// TwinCAT 3 PLC project CNM_AssertionInterfaceTests
// Title: CNM_AssertionInterfaceTests
// Company: ekvip automation GmbH
// Author: boez & ajum
// ProjectVersion: 1.0.0.47
// Description: Foo bar baz
// ProgramVersion: 3.1.4026.16
// libraries:
//   CNM_AbstractObject, * (ekvip automation GmbH)
//   CNM_AssertionInterfaceLib, * (ekvip automation GmbH)
//   CNM_ReturnTypes, * (ekvip automation GmbH)
//   Tc2_CncBase, * (Beckhoff Automation GmbH)
//   Tc2_CncHli, * (Beckhoff Automation GmbH)
//   Tc2_Standard, * (Beckhoff Automation GmbH)
//   Tc2_System, * (Beckhoff Automation GmbH)
//   Tc2_Utilities, * (Beckhoff Automation GmbH)
//   Tc3_Module, * (Beckhoff Automation GmbH)
//   TcUnit, * (www.tcunit.org)
// project tree:
//   AssertionTester/AssertionResult/interfaces/ IAssertorContainer.TcIO
//   AssertionTester/AssertionTests/BinaryAssertions/classes/ BinaryAssertionsTests.TcPOU, gfdfdfdvdfvdfvdfvfdv.TcPOU
//   AssertionTester/AssertionTests/BitNumberAssertions/classes/ XWordAssertionTests.TcPOU
//   AssertionTester/AssertionTests/classes/ AbstractAssertorTest.TcPOU
//   AssertionTester/AssertionTests/DateTimeAssertions/classes/ DTAssertionTests.TcPOU, DateAssertionTests.TcPOU, TODAssertionTests.TcPOU
//   AssertionTester/AssertionTests/FloatAssertions/classes/ RealAssertionTests.TcPOU, LRealAssertionTests.TcPOU
//   AssertionTester/AssertionTests/FloatAssertions/types/structs/ LRealTestParameter.TcDUT
//   AssertionTester/AssertionTests/IntegerAssertions/classes/ DintAssertionTests.TcPOU, IntAssertionTests.TcPOU, LintAssertionTests.TcPOU, SintAssertionTests.TcPOU, UdintAssertionTests.TcPOU, UintAssertionTests.TcPOU, UlintAssertionTests.TcPOU, UsintAssertionTests.TcPOU, UxintAssertionTests.TcPOU, XintAssertionTests.TcPOU
//   AssertionTester/AssertionTests/PointerAssertions/ PointerAssertionsTests.TcPOU
//   AssertionTester/AssertionTests/StringAssertions/InputStructs/common/ AnyTestString.TcDUT, StringType.TcDUT
//   AssertionTester/AssertionTests/StringAssertions/InputStructs/containsStr/ containsDataStr.TcDUT
//   AssertionTester/AssertionTests/StringAssertions/InputStructs/isEmptyStr/ isEmptyDataStr.TcDUT
//   AssertionTester/AssertionTests/StringAssertions/InputStructs/isEqualStr/ isEqualToDataStr.TcDUT
//   AssertionTester/AssertionTests/StringAssertions/InputStructs/isLenghtBetweenStr/ IsLengthBetweenBasicData.TcDUT
//   AssertionTester/AssertionTests/StringAssertions/InputStructs/isLenghtStr/ FunctionType.TcDUT, IsLengthBasicData.TcDUT, StringTestDataIsLength.TcDUT, TypeToTest.TcDUT
//   AssertionTester/AssertionTests/StringAssertions/ StringAssertionTests.TcPOU
//   AssertionTester/AssertionTests/StringAssertions/TestDataSets/ containsNoTestDataSet.TcGVL, containsTestDataSet.TcGVL, endsWithDataSet.TcGVL, isEmptyTestDataSet.TcGVL, isEqualToTestDataSet.TcGVL, IsLengthBetweenDataSet.TcGVL, IsLengthTestDataSet.TcGVL, isNotEmtyTestDataSet.TcGVL, isNotEqualToTestDataSet.TcGVL, startsWithDataSet.TcGVL
//   AssertionTester/AssertionTests/TimeAssertions/ TimeAssertionsTests.TcPOU
//   AssertionTester/classes/ AssertionTester.TcPOU
//   AssertionTester/functions/ ArrayOfMessageStringToString.TcPOU
//   AssertionTester/interfaces/ IAttachAssertorContainer.TcIO
//   Project Information/ F_GetCompany.TcPOU, F_GetTitle.TcPOU, F_GetVersion.TcPOU
//   Version/ Global_Version.TcGVL

// ---- AssertionTester/AssertionTests/FloatAssertions/types/structs/LRealTestParameter.TcDUT
(*

short summary
=================
this is just a helper type, the TwinCAT function LREAL_TO_STRING
throws an exception with the value 2.225073858507201e-308. 
since there is no big integer arithmetic at TwinCAT 
it's not in the scope of the test library to implement a doubleToString.
This data type contains just a LREAL value and it's string representation.

.. <legal notes>

legal notes
=================
| SPDX-FileCopyrightText: © 2022 ekvip automation GmbH <info@ekvip.de>
| SPDX-License-Identifier: Apache-2.0
| For details check: Apache-2.0_

.. _Apache-2.0: https://www.apache.org/licenses/LICENSE-2.0

.. </legal notes>

type members
======================

*)

TYPE LRealTestParameter :
STRUCT
	(* just the value to test *)
	value		:LREAL;
	(* string representation of ``value`` *)
	asString	:Tc2_System.T_MaxString;
END_STRUCT
END_TYPE

// ---- AssertionTester/AssertionTests/StringAssertions/InputStructs/common/AnyTestString.TcDUT
(*

short summary
=============

.. <legal notes>

legal notes
=================
| SPDX-FileCopyrightText: © 2023 ekvip automation GmbH <info@ekvip.de>
| SPDX-License-Identifier: Apache-2.0
| For details check: Apache-2.0_

.. _Apache-2.0: https://www.apache.org/licenses/LICENSE-2.0

.. </legal notes>

*)

{warning 'header is generated please add your documentation'}
TYPE AnyTestString :
STRUCT
	wstringToTest	:WSTRING(300);
	stringToTest	:STRING(600);
END_STRUCT
END_TYPE

// ---- AssertionTester/AssertionTests/StringAssertions/InputStructs/common/StringType.TcDUT
(*

short summary
=============

.. <legal notes>

legal notes
=================
| SPDX-FileCopyrightText: © 2023 ekvip automation GmbH <info@ekvip.de>
| SPDX-License-Identifier: Apache-2.0
| For details check: Apache-2.0_

.. _Apache-2.0: https://www.apache.org/licenses/LICENSE-2.0

.. </legal notes>

enumeration values
==================

*)

{warning 'header is generated please add your documentation'}
{attribute 'qualified_only'}
{attribute 'strict'}
{attribute 'to_string'}
TYPE StringType :
(
	ASCII_STRING := 0,
	UTF16STRING  := 1
)USINT;
END_TYPE

// ---- AssertionTester/AssertionTests/StringAssertions/InputStructs/containsStr/containsDataStr.TcDUT
(*

short summary
=============

.. <legal notes>

legal notes
=================
| SPDX-FileCopyrightText: © 2023 ekvip automation GmbH <info@ekvip.de>
| SPDX-License-Identifier: Apache-2.0
| For details check: Apache-2.0_

.. _Apache-2.0: https://www.apache.org/licenses/LICENSE-2.0

.. </legal notes>

*)

{warning 'header is generated please add your documentation'}
TYPE containsDataStr :
STRUCT
	StringToTest		: STRING;
	WStringToTest 		: WSTRING;
	StringToContain 	: STRING;
	WStringToContain	: WSTRING;
	IgnoreCases			: BOOL;
	Trim 				: BOOL;
	ExpectedResult  	: BOOL;
	typeToTest      	: TypeToTest;		
END_STRUCT
END_TYPE

// ---- AssertionTester/AssertionTests/StringAssertions/InputStructs/isEmptyStr/isEmptyDataStr.TcDUT
(*

short summary
=============

.. <legal notes>

legal notes
=================
| SPDX-FileCopyrightText: © 2023 ekvip automation GmbH <info@ekvip.de>
| SPDX-License-Identifier: Apache-2.0
| For details check: Apache-2.0_

.. _Apache-2.0: https://www.apache.org/licenses/LICENSE-2.0

.. </legal notes>

*)

{warning 'header is generated please add your documentation'}
TYPE isEmptyDataStr :
STRUCT
	StringToTest		: STRING;
	WStringToTest 		: WSTRING;
	ExpectedResult  	: BOOL;
	typeToTest      	: TypeToTest;		
END_STRUCT
END_TYPE

// ---- AssertionTester/AssertionTests/StringAssertions/InputStructs/isEqualStr/isEqualToDataStr.TcDUT
(*

short summary
=============

.. <legal notes>

legal notes
=================
| SPDX-FileCopyrightText: © 2023 ekvip automation GmbH <info@ekvip.de>
| SPDX-License-Identifier: Apache-2.0
| For details check: Apache-2.0_

.. _Apache-2.0: https://www.apache.org/licenses/LICENSE-2.0

.. </legal notes>

*)

{warning 'header is generated please add your documentation'}
TYPE isEqualToDataStr :
STRUCT
	StringToTest		: STRING;
	WStringToTest 		: WSTRING;
	EqualToString		: STRING;
	EqualToWString 		: WSTRING;
	IgnoreCases			: BOOL;
	ExpectedResult  	: BOOL;
	typeToTest      	: TypeToTest;		
END_STRUCT
END_TYPE

// ---- AssertionTester/AssertionTests/StringAssertions/InputStructs/isLenghtBetweenStr/IsLengthBetweenBasicData.TcDUT
(*

short summary
=============

.. <legal notes>

legal notes
=================
| SPDX-FileCopyrightText: © 2023 ekvip automation GmbH <info@ekvip.de>
| SPDX-License-Identifier: Apache-2.0
| For details check: Apache-2.0_

.. _Apache-2.0: https://www.apache.org/licenses/LICENSE-2.0

.. </legal notes>

*)

{warning 'header is generated please add your documentation'}
TYPE IsLengthBetweenBasicData :
STRUCT
	StringToTest	: STRING;
	WStringToTest	: WSTRING;
	ExpectedResult  : BOOL;
	maxLength		: USINT;
	minLength		: USINT; 
	typeToTest      : TypeToTest;  
END_STRUCT
END_TYPE

// ---- AssertionTester/AssertionTests/StringAssertions/InputStructs/isLenghtStr/FunctionType.TcDUT
(*

short summary
=============

.. <legal notes>

legal notes
=================
| SPDX-FileCopyrightText: © 2023 ekvip automation GmbH <info@ekvip.de>
| SPDX-License-Identifier: Apache-2.0
| For details check: Apache-2.0_

.. _Apache-2.0: https://www.apache.org/licenses/LICENSE-2.0

.. </legal notes>

enumeration values
==================

*)

{warning 'header is generated please add your documentation'}
{attribute 'qualified_only'}
{attribute 'strict'}
{attribute 'to_string'}
TYPE FunctionType :
(
	EXACT 	:= 0,
	MAXIMUM := 1,
	MINIMUM	:= 2 
);
END_TYPE

// ---- AssertionTester/AssertionTests/StringAssertions/InputStructs/isLenghtStr/IsLengthBasicData.TcDUT
(*

short summary
=============

.. <legal notes>

legal notes
=================
| SPDX-FileCopyrightText: © 2023 ekvip automation GmbH <info@ekvip.de>
| SPDX-License-Identifier: Apache-2.0
| For details check: Apache-2.0_

.. _Apache-2.0: https://www.apache.org/licenses/LICENSE-2.0

.. </legal notes>

*)

{warning 'header is generated please add your documentation'}
TYPE IsLengthBasicData :
STRUCT
	StringToTest	: STRING;
	WStringToTest	: WSTRING;
	ExpectedResult  : BOOL;
	ExpectedLength	: UDINT; 
	FuncType		: FunctionType;
	typeToTest      : TypeToTest;  	
END_STRUCT
END_TYPE

// ---- AssertionTester/AssertionTests/StringAssertions/InputStructs/isLenghtStr/StringTestDataIsLength.TcDUT
(*

short summary
=============

.. <legal notes>

legal notes
=================
| SPDX-FileCopyrightText: © 2023 ekvip automation GmbH <info@ekvip.de>
| SPDX-License-Identifier: Apache-2.0
| For details check: Apache-2.0_

.. _Apache-2.0: https://www.apache.org/licenses/LICENSE-2.0

.. </legal notes>

*)

{warning 'header is generated please add your documentation'}
TYPE StringTestDataIsLength :
STRUCT
	testString		: AnyTestString ;
	expectedLength	: UDINT;
	stringType		: StringType;
	message			: STRING;
	expectedResult	: BOOL;
    funcType		: FunctionType;     
END_STRUCT
END_TYPE

// ---- AssertionTester/AssertionTests/StringAssertions/InputStructs/isLenghtStr/TypeToTest.TcDUT
(*

short summary
=============

.. <legal notes>

legal notes
=================
| SPDX-FileCopyrightText: © 2023 ekvip automation GmbH <info@ekvip.de>
| SPDX-License-Identifier: Apache-2.0
| For details check: Apache-2.0_

.. _Apache-2.0: https://www.apache.org/licenses/LICENSE-2.0

.. </legal notes>

enumeration values
==================

*)

{warning 'header is generated please add your documentation'}
{attribute 'qualified_only'}
{attribute 'strict'}
TYPE TypeToTest :
(
	TEST_STRING 	:= 0,
	TEST_WSTRING 	:= 1
);
END_TYPE

// ---- AssertionTester/AssertionTests/StringAssertions/TestDataSets/containsNoTestDataSet.TcGVL
(*

short summary
=============

.. <legal notes>

legal notes
=================
| SPDX-FileCopyrightText: © 2023 ekvip automation GmbH <info@ekvip.de>
| SPDX-License-Identifier: Apache-2.0
| For details check: Apache-2.0_

.. _Apache-2.0: https://www.apache.org/licenses/LICENSE-2.0

.. </legal notes>

*)

{warning 'header is generated please add your documentation'}
{attribute 'qualified_only'}
VAR_GLOBAL CONSTANT
	SIZE_OF_CONTAINSNO_DATASET:USINT := 21;
END_VAR

VAR_GLOBAL
	containsNoDataSetCommon : ARRAY[0..SIZE_OF_CONTAINSNO_DATASET] OF containsDataStr := [
		
		// test number 0
		(	StringToTest		:= 'hello',
		  	WStringToTest 		:= "Hello",
			StringToContain 	:= 'h',
			WStringToContain	:= "h",
			IgnoreCases			:= TRUE,
			ExpectedResult  	:= TRUE,
			typeToTest      	:= TypeToTest.TEST_STRING	),
		
		// test number 1	
		(	StringToTest		:= 'hello',
		  	WStringToTest 		:= "Hello",
			StringToContain 	:= 'h',
			WStringToContain	:= "h",
			IgnoreCases			:= TRUE,
			ExpectedResult  	:= TRUE,
			typeToTest      	:= TypeToTest.TEST_WSTRING	),
		
		// test number 2		
		(	StringToTest		:= 'дивный новый мир',
		  	WStringToTest 		:= "дивный новый мир",
			StringToContain 	:= 'нов',
			WStringToContain	:= "нов",
			IgnoreCases			:= TRUE,
			ExpectedResult  	:= TRUE,
			typeToTest      	:= TypeToTest.TEST_WSTRING	),

		// test number 3				
		(	StringToTest		:= 'дивный новый мир',
		  	WStringToTest 		:= "дивный новый мир",
			StringToContain 	:= 'ноa',
			WStringToContain	:= "ноa",
			IgnoreCases			:= TRUE,
			ExpectedResult  	:= FALSE,
			typeToTest      	:= TypeToTest.TEST_WSTRING	),

		// test number 4				
		(	StringToTest		:= 'дивный новый мир',
		  	WStringToTest 		:= "дивный новый мир",
			StringToContain 	:= 'нов',
			WStringToContain	:= "нов",
			IgnoreCases			:= TRUE,
			ExpectedResult  	:= TRUE,
			typeToTest      	:= TypeToTest.TEST_STRING	),
	
		// test number 5			
		(	StringToTest		:= 'дивный новый мир',
		  	WStringToTest 		:= "дивный новый мир",
			StringToContain 	:= 'ноa',
			WStringToContain	:= "ноa",
			IgnoreCases			:= TRUE,
			ExpectedResult  	:= FALSE,
			typeToTest      	:= TypeToTest.TEST_STRING	),
			
		// test number 6			
		(	StringToTest		:= '',
		  	WStringToTest 		:= "",
			StringToContain 	:= ' ',
			WStringToContain	:= " ",
			IgnoreCases			:= TRUE,
			ExpectedResult  	:= FALSE,
			typeToTest      	:= TypeToTest.TEST_STRING	),
			
		// test number 7			
		(	StringToTest		:= '',
		  	WStringToTest 		:= "",
			StringToContain 	:= ' ',
			WStringToContain	:= " ",
			IgnoreCases			:= TRUE,
			ExpectedResult  	:= FALSE,
			typeToTest      	:= TypeToTest.TEST_WSTRING	),
			
		// test number 8			
		(	StringToTest		:= ' ',
		  	WStringToTest 		:= " ",
			StringToContain 	:= ' ',
			WStringToContain	:= " ",
			IgnoreCases			:= TRUE,
			ExpectedResult  	:= TRUE,
			typeToTest      	:= TypeToTest.TEST_STRING	),
			
		// test number 9			
		(	StringToTest		:= ' ',
		  	WStringToTest 		:= " ",
			StringToContain 	:= ' ',
			WStringToContain	:= " ",
			IgnoreCases			:= TRUE,
			ExpectedResult  	:= TRUE,
			typeToTest      	:= TypeToTest.TEST_WSTRING	),
			
		// test number 10			
		(	StringToTest		:= ' ',
		  	WStringToTest 		:= " ",
			StringToContain 	:= ' ',
			WStringToContain	:= " ",
			IgnoreCases			:= TRUE,
			ExpectedResult  	:= TRUE,
			typeToTest      	:= TypeToTest.TEST_STRING	),
			
		// test number 11			
		(	StringToTest		:= 'Brave new World',
		  	WStringToTest 		:= "Brave new World",
			StringToContain 	:= 'brave',
			WStringToContain	:= "brave",
			IgnoreCases			:= FALSE,
			ExpectedResult  	:= FALSE,
			typeToTest      	:= TypeToTest.TEST_WSTRING	),
			
		// test number 12			
		(	StringToTest		:= 'Brave new World',
		  	WStringToTest 		:= "Brave new World",
			StringToContain 	:= 'brave',
			WStringToContain	:= "brave",
			IgnoreCases			:= FALSE,
			ExpectedResult  	:= FALSE,
			typeToTest      	:= TypeToTest.TEST_WSTRING	),
			
		// test number 13			
		(	StringToTest		:= 'Brave new World',
		  	WStringToTest 		:= "Brave new World",
			StringToContain 	:= 'brave',
			WStringToContain	:= "brave",
			IgnoreCases			:= TRUE,
			ExpectedResult  	:= TRUE,
			typeToTest      	:= TypeToTest.TEST_WSTRING	),
			
		// test number 14			
		(	StringToTest		:= 'Brave new World',
		  	WStringToTest 		:= "Brave new World",
			StringToContain 	:= 'brave',
			WStringToContain	:= "brave",
			IgnoreCases			:= TRUE,
			ExpectedResult  	:= TRUE,
			typeToTest      	:= TypeToTest.TEST_WSTRING	),
			
		// test number 15			
		(	StringToTest		:= '²345',
		  	WStringToTest 		:= "²345",
			StringToContain 	:= '2',
			WStringToContain	:= "2",
			IgnoreCases			:= TRUE,
			ExpectedResult  	:= FALSE,
			typeToTest      	:= TypeToTest.TEST_STRING	),
			
		// test number 16			
		(	StringToTest		:= '2345',
		  	WStringToTest 		:= "²345",
			StringToContain 	:= '2',
			WStringToContain	:= "2",
			IgnoreCases			:= TRUE,
			ExpectedResult  	:= FALSE,
			typeToTest      	:= TypeToTest.TEST_WSTRING	),
			
		// test number 17			
		(	StringToTest		:= '²345',
		  	WStringToTest 		:= "²345",
			StringToContain 	:= '2',
			WStringToContain	:= "2",
			IgnoreCases			:= FALSE,
			ExpectedResult  	:= FALSE,
			typeToTest      	:= TypeToTest.TEST_STRING	),
			
		// test number 18			
		(	StringToTest		:= '²345',
		  	WStringToTest 		:= "²345",
			StringToContain 	:= '2',
			WStringToContain	:= "2",
			IgnoreCases			:= FALSE,
			ExpectedResult  	:= FALSE,
			typeToTest      	:= TypeToTest.TEST_WSTRING	),
			
		// test number 19			
		(	StringToTest		:= '',
		  	WStringToTest 		:= "👪",
			StringToContain 	:= '',
			WStringToContain	:= "👪",
			IgnoreCases			:= FALSE,
			ExpectedResult  	:= TRUE,
			typeToTest      	:= TypeToTest.TEST_WSTRING	),
			
		// test number 20			
		(	StringToTest		:= ' hello world ',
		  	WStringToTest 		:= " hello world ",
			StringToContain 	:= '  ',
			WStringToContain	:= "  ",
			IgnoreCases			:= FALSE,
			ExpectedResult  	:= FALSE,
			typeToTest      	:= TypeToTest.TEST_WSTRING	),
			
		// test number 21			
		(	StringToTest		:= ' hello world ',
		  	WStringToTest 		:= " hello world ",
			StringToContain 	:= '  ',
			WStringToContain	:= "  ",
			IgnoreCases			:= FALSE,
			ExpectedResult  	:= FALSE,
			typeToTest      	:= TypeToTest.TEST_STRING	)
			
		
			
		

	];
END_VAR

// ---- AssertionTester/AssertionTests/StringAssertions/TestDataSets/containsTestDataSet.TcGVL
(*

short summary
=============

.. <legal notes>

legal notes
=================
| SPDX-FileCopyrightText: © 2023 ekvip automation GmbH <info@ekvip.de>
| SPDX-License-Identifier: Apache-2.0
| For details check: Apache-2.0_

.. _Apache-2.0: https://www.apache.org/licenses/LICENSE-2.0

.. </legal notes>

*)

{warning 'header is generated please add your documentation'}
{attribute 'qualified_only'}
VAR_GLOBAL CONSTANT
	SIZE_OF_CONTAINS_DATASET:USINT := 23;
END_VAR

VAR_GLOBAL
	containsDataSetCommon : ARRAY[0..SIZE_OF_CONTAINS_DATASET] OF containsDataStr := [
		// test number 0
		(	StringToTest		:= 'hello',
		  	WStringToTest 		:= "Hello",
			StringToContain 	:= 'h',
			WStringToContain	:= "h",
			IgnoreCases			:= TRUE,
			ExpectedResult  	:= FALSE,
			typeToTest      	:= TypeToTest.TEST_STRING	),
		
		// test number 1	
		(	StringToTest		:= 'hello',
		  	WStringToTest 		:= "Hello",
			StringToContain 	:= 'h',
			WStringToContain	:= "h",
			IgnoreCases			:= TRUE,
			ExpectedResult  	:= FALSE,
			typeToTest      	:= TypeToTest.TEST_WSTRING	),
		
		// test number 2		
		(	StringToTest		:= 'дивный новый мир',
		  	WStringToTest 		:= "дивный новый мир",
			StringToContain 	:= 'нов',
			WStringToContain	:= "нов",
			IgnoreCases			:= TRUE,
			ExpectedResult  	:= FALSE,
			typeToTest      	:= TypeToTest.TEST_WSTRING	),

		// test number 3				
		(	StringToTest		:= 'дивный новый мир',
		  	WStringToTest 		:= "дивный новый мир",
			StringToContain 	:= 'ноa',
			WStringToContain	:= "ноa",
			IgnoreCases			:= TRUE,
			ExpectedResult  	:= TRUE,
			typeToTest      	:= TypeToTest.TEST_WSTRING	),

		// test number 4				
		(	StringToTest		:= 'дивный новый мир',
		  	WStringToTest 		:= "дивный новый мир",
			StringToContain 	:= 'нов',
			WStringToContain	:= "нов",
			IgnoreCases			:= TRUE,
			ExpectedResult  	:= FALSE,
			typeToTest      	:= TypeToTest.TEST_STRING	),
	
		// test number 5			
		(	StringToTest		:= 'дивный новый мир',
		  	WStringToTest 		:= "дивный новый мир",
			StringToContain 	:= 'ноa',
			WStringToContain	:= "ноa",
			IgnoreCases			:= TRUE,
			ExpectedResult  	:= TRUE,
			typeToTest      	:= TypeToTest.TEST_STRING	),
			
		// test number 6			
		(	StringToTest		:= '',
		  	WStringToTest 		:= "",
			StringToContain 	:= ' ',
			WStringToContain	:= " ",
			IgnoreCases			:= TRUE,
			ExpectedResult  	:= TRUE,
			typeToTest      	:= TypeToTest.TEST_STRING	),
			
		// test number 7			
		(	StringToTest		:= '',
		  	WStringToTest 		:= "",
			StringToContain 	:= ' ',
			WStringToContain	:= " ",
			IgnoreCases			:= TRUE,
			ExpectedResult  	:= TRUE,
			typeToTest      	:= TypeToTest.TEST_WSTRING	),
			
		// test number 8			
		(	StringToTest		:= ' ',
		  	WStringToTest 		:= " ",
			StringToContain 	:= ' ',
			WStringToContain	:= " ",
			IgnoreCases			:= TRUE,
			ExpectedResult  	:= FALSE,
			typeToTest      	:= TypeToTest.TEST_STRING	),
			
		// test number 9			
		(	StringToTest		:= ' ',
		  	WStringToTest 		:= " ",
			StringToContain 	:= ' ',
			WStringToContain	:= " ",
			IgnoreCases			:= TRUE,
			ExpectedResult  	:= FALSE,
			typeToTest      	:= TypeToTest.TEST_WSTRING	),
			
		// test number 10			
		(	StringToTest		:= ' ',
		  	WStringToTest 		:= " ",
			StringToContain 	:= ' ',
			WStringToContain	:= " ",
			IgnoreCases			:= TRUE,
			ExpectedResult  	:= FALSE,
			typeToTest      	:= TypeToTest.TEST_STRING	),
			
		// test number 11			
		(	StringToTest		:= 'Brave new World',
		  	WStringToTest 		:= "Brave new World",
			StringToContain 	:= 'brave',
			WStringToContain	:= "brave",
			IgnoreCases			:= FALSE,
			ExpectedResult  	:= TRUE,
			typeToTest      	:= TypeToTest.TEST_WSTRING	),
			
		// test number 12			
		(	StringToTest		:= 'Brave new World',
		  	WStringToTest 		:= "Brave new World",
			StringToContain 	:= 'brave',
			WStringToContain	:= "brave",
			IgnoreCases			:= FALSE,
			ExpectedResult  	:= TRUE,
			typeToTest      	:= TypeToTest.TEST_WSTRING	),
			
		// test number 13			
		(	StringToTest		:= 'Brave new World',
		  	WStringToTest 		:= "Brave new World",
			StringToContain 	:= 'brave',
			WStringToContain	:= "brave",
			IgnoreCases			:= TRUE,
			ExpectedResult  	:= FALSE,
			typeToTest      	:= TypeToTest.TEST_WSTRING	),
			
		// test number 14			
		(	StringToTest		:= 'Brave new World',
		  	WStringToTest 		:= "Brave new World",
			StringToContain 	:= 'brave',
			WStringToContain	:= "brave",
			IgnoreCases			:= TRUE,
			ExpectedResult  	:= FALSE,
			typeToTest      	:= TypeToTest.TEST_WSTRING	),
			
		// test number 15			
		(	StringToTest		:= '²345',
		  	WStringToTest 		:= "²345",
			StringToContain 	:= '2',
			WStringToContain	:= "2",
			IgnoreCases			:= TRUE,
			ExpectedResult  	:= TRUE,
			typeToTest      	:= TypeToTest.TEST_STRING	),
			
		// test number 16			
		(	StringToTest		:= '2345',
		  	WStringToTest 		:= "²345",
			StringToContain 	:= '2',
			WStringToContain	:= "2",
			IgnoreCases			:= TRUE,
			ExpectedResult  	:= TRUE,
			typeToTest      	:= TypeToTest.TEST_WSTRING	),
			
		// test number 17			
		(	StringToTest		:= '²345',
		  	WStringToTest 		:= "²345",
			StringToContain 	:= '2',
			WStringToContain	:= "2",
			IgnoreCases			:= FALSE,
			ExpectedResult  	:= TRUE,
			typeToTest      	:= TypeToTest.TEST_STRING	),
			
		// test number 18			
		(	StringToTest		:= '²345',
		  	WStringToTest 		:= "²345",
			StringToContain 	:= '2',
			WStringToContain	:= "2",
			IgnoreCases			:= FALSE,
			ExpectedResult  	:= TRUE,
			typeToTest      	:= TypeToTest.TEST_WSTRING	),
			
		// test number 19			
		(	StringToTest		:= '',
		  	WStringToTest 		:= "👪",
			StringToContain 	:= '',
			WStringToContain	:= "👪",
			IgnoreCases			:= FALSE,
			ExpectedResult  	:= FALSE,
			typeToTest      	:= TypeToTest.TEST_WSTRING	),
			
		// test number 20			
		(	StringToTest		:= ' hello world ',
		  	WStringToTest 		:= " hello world ",
			StringToContain 	:= '  ',
			WStringToContain	:= "  ",
			IgnoreCases			:= FALSE,
			ExpectedResult  	:= TRUE,
			typeToTest      	:= TypeToTest.TEST_WSTRING	),
			
		// test number 21			
		(	StringToTest		:= ' hello world ',
		  	WStringToTest 		:= " hello world ",
			StringToContain 	:= '  ',
			WStringToContain	:= "  ",
			IgnoreCases			:= FALSE,
			ExpectedResult  	:= TRUE,
			typeToTest      	:= TypeToTest.TEST_STRING	),
			
		// test number 22			
		(	StringToTest		:= '',
		  	WStringToTest 		:= "∛",
			StringToContain 	:= '',
			WStringToContain	:= "√∛∜",
			IgnoreCases			:= FALSE,
			ExpectedResult  	:= TRUE,
			typeToTest      	:= TypeToTest.TEST_WSTRING	),
			
		// test number 23			
		(	StringToTest		:= '',
		  	WStringToTest 		:= "∭∝√∛∜",
			StringToContain 	:= '',
			WStringToContain	:= "∬",
			IgnoreCases			:= FALSE,
			ExpectedResult  	:= TRUE,
			typeToTest      	:= TypeToTest.TEST_WSTRING	)

					
						
	];
END_VAR

// ---- AssertionTester/AssertionTests/StringAssertions/TestDataSets/endsWithDataSet.TcGVL
(*

short summary
=============

.. <legal notes>

legal notes
=================
| SPDX-FileCopyrightText: © 2023 ekvip automation GmbH <info@ekvip.de>
| SPDX-License-Identifier: Apache-2.0
| For details check: Apache-2.0_

.. _Apache-2.0: https://www.apache.org/licenses/LICENSE-2.0

.. </legal notes>

*)

{warning 'header is generated please add your documentation'}
{attribute 'qualified_only'}
VAR_GLOBAL CONSTANT
	SIZE_OF_ENDSWITH_DATASET:USINT := 18;
END_VAR

VAR_GLOBAL
	endsWithDataSetCommon : ARRAY[0..SIZE_OF_ENDSWITH_DATASET] OF containsDataStr := [
		
		// Test number 0
		(	StringToTest		:= 'HellO',
		  	WStringToTest 		:= "HellO",
			StringToContain 	:= 'lo',
			WStringToContain	:= "lo",
			IgnoreCases			:= TRUE,
			Trim 				:= FALSE,
			ExpectedResult  	:= FALSE,
			typeToTest      	:= TypeToTest.TEST_STRING	),
		
		// Test number 1	
		(	StringToTest		:= 'HellO',
		  	WStringToTest 		:= "HellO",
			StringToContain 	:= 'lo',
			WStringToContain	:= "lo",
			IgnoreCases			:= TRUE,
			Trim 				:= FALSE,
			ExpectedResult  	:= FALSE,
			typeToTest      	:= TypeToTest.TEST_WSTRING	),
		
		// Test number 2	
		(	StringToTest		:= 'Hello',
		  	WStringToTest 		:= "Hello",
			StringToContain 	:= 'LO',
			WStringToContain	:= "LO",
			IgnoreCases			:= FALSE,
			Trim 				:= FALSE,
			ExpectedResult  	:= TRUE,
			typeToTest      	:= TypeToTest.TEST_STRING	),

		// Test number 3			
		(	StringToTest		:= 'Hello',
		  	WStringToTest 		:= "Hello",
			StringToContain 	:= 'LO',
			WStringToContain	:= "LO",
			IgnoreCases			:= FALSE,
			Trim 				:= FALSE,
			ExpectedResult  	:= TRUE,
			typeToTest      	:= TypeToTest.TEST_WSTRING	),
			
		// Test number 4	
		(	StringToTest		:= 'Hello ',
		  	WStringToTest 		:= "Hello ",
			StringToContain 	:= 'lo',
			WStringToContain	:= "lo",
			IgnoreCases			:= FALSE,
			Trim 				:= TRUE,
			ExpectedResult  	:= FALSE,
			typeToTest      	:= TypeToTest.TEST_STRING	),

		// Test number 5			
		(	StringToTest		:= 'Hello ',
		  	WStringToTest 		:= "Hello ",
			StringToContain 	:= 'lo',
			WStringToContain	:= "lo",
			IgnoreCases			:= FALSE,
			Trim 				:= TRUE,
			ExpectedResult  	:= FALSE,
			typeToTest      	:= TypeToTest.TEST_WSTRING	),
			
		// Test number 6	
		(	StringToTest		:= 'Kind and evil',
		  	WStringToTest 		:= "Добро и зло",
			StringToContain 	:= 'evil',
			WStringToContain	:= "зло",
			IgnoreCases			:= FALSE,
			Trim 				:= FALSE,
			ExpectedResult  	:= FALSE,
			typeToTest      	:= TypeToTest.TEST_STRING	),

		// Test number 7			
		(	StringToTest		:= 'Kind and evil',
		  	WStringToTest 		:= "Добро и зло",
			StringToContain 	:= 'evil',
			WStringToContain	:= "зло",
			IgnoreCases			:= FALSE,
			Trim 				:= FALSE,
			ExpectedResult  	:= FALSE,
			typeToTest      	:= TypeToTest.TEST_WSTRING	),
			
		// Test number 8	
		(	StringToTest		:= 'Kind and evil',
		  	WStringToTest 		:= "Добро и зло",
			StringToContain 	:= 'evi',
			WStringToContain	:= "зл",
			IgnoreCases			:= FALSE,
			Trim 				:= FALSE,
			ExpectedResult  	:= TRUE,
			typeToTest      	:= TypeToTest.TEST_STRING	),

		// Test number 9			
		(	StringToTest		:= 'Kind and evil',
		  	WStringToTest 		:= "Добро и зло",
			StringToContain 	:= 'evi',
			WStringToContain	:= "зл",
			IgnoreCases			:= FALSE,
			Trim 				:= FALSE,
			ExpectedResult  	:= TRUE,
			typeToTest      	:= TypeToTest.TEST_WSTRING	),
			
		// Test number 10	
		(	StringToTest		:= 'Kind and evil',
		  	WStringToTest 		:= "Добро и зло",
			StringToContain 	:= 'evil',
			WStringToContain	:= "Зло",
			IgnoreCases			:= TRUE,
			Trim 				:= FALSE,
			ExpectedResult  	:= FALSE,
			typeToTest      	:= TypeToTest.TEST_STRING	),

		// Test number 11			
		(	StringToTest		:= 'Kind and evil',
		  	WStringToTest 		:= "Добро и зло",
			StringToContain 	:= 'evil',
			WStringToContain	:= "Зло",
			IgnoreCases			:= TRUE,
			Trim 				:= FALSE,
			ExpectedResult  	:= FALSE,
			typeToTest      	:= TypeToTest.TEST_WSTRING	),
			
		// Test number 12	
		(	StringToTest		:= ' Kind and evil ',
		  	WStringToTest 		:= " Добро и зло ",
			StringToContain 	:= 'evil',
			WStringToContain	:= "зло",
			IgnoreCases			:= TRUE,
			Trim 				:= TRUE,
			ExpectedResult  	:= FALSE,
			typeToTest      	:= TypeToTest.TEST_STRING	),

		// Test number 13			
		(	StringToTest		:= ' Kind and evil ',
		  	WStringToTest 		:= " Добро и зло ",
			StringToContain 	:= 'evil',
			WStringToContain	:= "зло",
			IgnoreCases			:= TRUE,
			Trim 				:= TRUE,
			ExpectedResult  	:= FALSE,
			typeToTest      	:= TypeToTest.TEST_WSTRING	),
			
		// Test number 14			
		(	StringToTest		:= '',
		  	WStringToTest 		:= " 🧛 ",
			StringToContain 	:= '',
			WStringToContain	:= "🧛",
			IgnoreCases			:= TRUE,
			Trim 				:= TRUE,
			ExpectedResult  	:= FALSE,
			typeToTest      	:= TypeToTest.TEST_WSTRING	),
			
		// Test number 15			
		(	StringToTest		:= '',
		  	WStringToTest 		:= " 🧛 ",
			StringToContain 	:= '',
			WStringToContain	:= "🧛",
			IgnoreCases			:= TRUE,
			Trim 				:= FALSE,
			ExpectedResult  	:= TRUE,
			typeToTest      	:= TypeToTest.TEST_WSTRING	),

		// Test number 16			
		(	StringToTest		:= '',
		  	WStringToTest 		:= "🧛",
			StringToContain 	:= '',
			WStringToContain	:= "🧛",
			IgnoreCases			:= FALSE,
			Trim 				:= FALSE,
			ExpectedResult  	:= FALSE,
			typeToTest      	:= TypeToTest.TEST_WSTRING	),
			
		// Test number 17			
		(	StringToTest		:= ' hello world ',
		  	WStringToTest 		:= " hello world ",
			StringToContain 	:= '  ',
			WStringToContain	:= "  ",
			IgnoreCases			:= TRUE,
			Trim 				:= FALSE,
			ExpectedResult  	:= TRUE,
			typeToTest      	:= TypeToTest.TEST_WSTRING	),

		// Test number 18			
		(	StringToTest		:= ' hello world ',
		  	WStringToTest 		:= " hello world ",
			StringToContain 	:= '  ',
			WStringToContain	:= "  ",
			IgnoreCases			:= TRUE,
			Trim 				:= FALSE,
			ExpectedResult  	:= TRUE,
			typeToTest      	:= TypeToTest.TEST_STRING	)
			
					

	];
END_VAR

// ---- AssertionTester/AssertionTests/StringAssertions/TestDataSets/isEmptyTestDataSet.TcGVL
(*

short summary
=============

.. <legal notes>

legal notes
=================
| SPDX-FileCopyrightText: © 2023 ekvip automation GmbH <info@ekvip.de>
| SPDX-License-Identifier: Apache-2.0
| For details check: Apache-2.0_

.. _Apache-2.0: https://www.apache.org/licenses/LICENSE-2.0

.. </legal notes>

*)

{warning 'header is generated please add your documentation'}
{attribute 'qualified_only'}
VAR_GLOBAL CONSTANT
	SIZE_OF_ISEMPTY_DATASET:USINT := 13;
END_VAR

VAR_GLOBAL
	isEmptyDataSetCommon : ARRAY[0..SIZE_OF_ISEMPTY_DATASET] OF isEmptyDataStr := [
		// test number 0
		(	StringToTest 	:= 'hello',
			WStringToTest 	:= "hello",
			ExpectedResult  := TRUE,
			typeToTest     	:= TypeToTest.TEST_STRING ),
		
		// test number 1
		(	StringToTest 	:= 'hello',
			WStringToTest 	:= "hello",
			ExpectedResult  := TRUE,
			typeToTest     	:= TypeToTest.TEST_STRING ),

		// test number 2
		(	StringToTest 	:= '',
			WStringToTest 	:= "",
			ExpectedResult  := FALSE,
			typeToTest     	:= TypeToTest.TEST_STRING ),		
		
		// test number 3
		(	StringToTest 	:= '',
			WStringToTest 	:= "",
			ExpectedResult  := FALSE,
			typeToTest     	:= TypeToTest.TEST_WSTRING ),	

		// test number 4
		(	StringToTest 	:= '   ',
			WStringToTest 	:= "   ",
			ExpectedResult  := TRUE,
			typeToTest     	:= TypeToTest.TEST_WSTRING ),

		// test number 5
		(	StringToTest 	:= '   ',
			WStringToTest 	:= "   ",
			ExpectedResult  := TRUE,
			typeToTest     	:= TypeToTest.TEST_STRING ),
			
		// test number 6
		(	StringToTest 	:= '   ',
			WStringToTest 	:= "नमस्ते",
			ExpectedResult  := TRUE,
			typeToTest     	:= TypeToTest.TEST_WSTRING ),
				
		// test number 7
		(	StringToTest 	:= 'мальчик или девочка',
			WStringToTest 	:= "мальчик или девочка",
			ExpectedResult  := TRUE,
			typeToTest     	:= TypeToTest.TEST_WSTRING ),
			
		// test number 8
		(	StringToTest 	:= 'мальчик или девочка',
			WStringToTest 	:= "мальчик или девочка",
			ExpectedResult  := TRUE,
			typeToTest     	:= TypeToTest.TEST_STRING ),
			
		// test number 9
		(	StringToTest 	:= '',
			WStringToTest 	:= "👨‍🔬 👩‍🎨 🧑‍🎨 👨‍🎨 👩‍🚒 🧑‍🚒 👨‍🚒 👩‍✈️ 🧑‍✈️ 👨‍✈️ 👩‍🚀",
			ExpectedResult  := TRUE,
			typeToTest     	:= TypeToTest.TEST_WSTRING ),
			
		// test number 10
		(	StringToTest 	:= 'QQQqqqq@@@@@%%%%',
			WStringToTest 	:= "QQQqqqq@@@@@%%%%",
			ExpectedResult  := TRUE,
			typeToTest     	:= TypeToTest.TEST_WSTRING ),

		// test number 11
		(	StringToTest 	:= '.',
			WStringToTest 	:= ".",
			ExpectedResult  := TRUE,
			typeToTest     	:= TypeToTest.TEST_WSTRING ),	

			
		// test number 12
		(	StringToTest 	:= 'QQQqqqq@@@@@%%%%',
			WStringToTest 	:= "QQQqqqq@@@@@%%%%",
			ExpectedResult  := TRUE,
			typeToTest     	:= TypeToTest.TEST_STRING ),

		// test number 13
		(	StringToTest 	:= '.',
			WStringToTest 	:= ".",
			ExpectedResult  := TRUE,
			typeToTest     	:= TypeToTest.TEST_STRING )			

	];
END_VAR

// ---- AssertionTester/AssertionTests/StringAssertions/TestDataSets/isEqualToTestDataSet.TcGVL
(*

short summary
=============

.. <legal notes>

legal notes
=================
| SPDX-FileCopyrightText: © 2023 ekvip automation GmbH <info@ekvip.de>
| SPDX-License-Identifier: Apache-2.0
| For details check: Apache-2.0_

.. _Apache-2.0: https://www.apache.org/licenses/LICENSE-2.0

.. </legal notes>

*)

{warning 'header is generated please add your documentation'}
{attribute 'qualified_only'}
VAR_GLOBAL CONSTANT
	SIZE_OF_ISEQUALTO_DATASET:USINT := 32;
END_VAR

VAR_GLOBAL
	isEqualToDataSetCommon : ARRAY[0..SIZE_OF_ISEQUALTO_DATASET] OF isEqualToDataStr := [
		// test number 0
		( 	StringToTest	:= 'hello',
			WStringToTest	:= "hello",
			EqualToString	:= 'hello',
			EqualToWString	:= "hello",
			IgnoreCases		:= FALSE,
			ExpectedResult	:= FALSE,
			typeToTest		:= TypeToTest.TEST_WSTRING ),

		// test number 1
		( 	StringToTest	:= 'Давным-давно, когда тигр курил',
			WStringToTest	:= "Давным-давно, когда тигр курил",
			EqualToString	:= 'Давным-давно, когда тигр курил',
			EqualToWString	:= "Давным-давно, когда тигр курил",
			IgnoreCases		:= FALSE,
			ExpectedResult	:= FALSE,
			typeToTest		:= TypeToTest.TEST_WSTRING ),
			
		// test number 2
		( 	StringToTest	:= 'לאנג צוריק ווען טיגערס פלעגן רייכערן',
			WStringToTest	:= "לאנג צוריק ווען טיגערס פלעגן רייכערן",
			EqualToString	:= 'לאנג צוריק ווען טיגערס פלעגן רייכערן',
			EqualToWString	:= "לאנג צוריק ווען טיגערס פלעגן רייכערן",
			IgnoreCases		:= FALSE,
			ExpectedResult	:= FALSE,
			typeToTest		:= TypeToTest.TEST_WSTRING ),
			
		// test number 3
		( 	StringToTest	:= 'Давным-давно, когда тигркурил',
			WStringToTest	:= "Давным-давно, когда тигркурил",
			EqualToString	:= 'Давным-давно, когда тигр курил',
			EqualToWString	:= "Давным-давно, когда тигр курил",
			IgnoreCases		:= FALSE,
			ExpectedResult	:= TRUE,
			typeToTest		:= TypeToTest.TEST_WSTRING ),
			
		// test number 4
		( 	StringToTest	:= 'לאנג צוריק ווען טיגערס פלעגןרייכערן',
			WStringToTest	:= "לאנג צוריק ווען טיגערס פלעגןרייכערן",
			EqualToString	:= 'לאנג צוריק ווען טיגערס פלעגן רייכערן',
			EqualToWString	:= "לאנג צוריק ווען טיגערס פלעגן רייכערן",
			IgnoreCases		:= FALSE,
			ExpectedResult	:= TRUE,
			typeToTest		:= TypeToTest.TEST_WSTRING ),
			
		// test number 5
		( 	StringToTest	:= 'לאנג צוריק ווען טיגערס פלעגןרייכערן',
			WStringToTest	:= "לאנג צוריק ווען טיגערס פלעגןרייכערן",
			EqualToString	:= 'לאנג צוריק ווע טיגערס פלעגןרייכערן',
			EqualToWString	:= "לאנג צוריק ווע טיגערס פלעגןרייכערן",
			IgnoreCases		:= FALSE,
			ExpectedResult	:= TRUE,
			typeToTest		:= TypeToTest.TEST_WSTRING ),
			
		// test number 6
		( 	StringToTest	:= '',
			WStringToTest	:= "",
			EqualToString	:= '',
			EqualToWString	:= "",
			IgnoreCases		:= FALSE,
			ExpectedResult	:= FALSE,
			typeToTest		:= TypeToTest.TEST_WSTRING ),
			
		// test number 7
		( 	StringToTest	:= ' ',
			WStringToTest	:= " ",
			EqualToString	:= '  ',
			EqualToWString	:= "  ",
			IgnoreCases		:= FALSE,
			ExpectedResult	:= TRUE,
			typeToTest		:= TypeToTest.TEST_WSTRING ),
			
		// test number 8
		( 	StringToTest	:= 'abc',
			WStringToTest	:= "abc",
			EqualToString	:= 'ABC',
			EqualToWString	:= "ABC",
			IgnoreCases		:= TRUE,
			ExpectedResult	:= FALSE,
			typeToTest		:= TypeToTest.TEST_WSTRING ),

		// test number 9
		( 	StringToTest	:= 'нефти и газа',
			WStringToTest	:= "нефти и газа",
			EqualToString	:= 'НЕФТИ И ГАЗА',
			EqualToWString	:= "НЕФТИ И ГАЗА",
			IgnoreCases		:= TRUE,
			ExpectedResult	:= FALSE,
			typeToTest		:= TypeToTest.TEST_WSTRING ),
		
		// test number 10
		( 	StringToTest	:= 'hello',
			WStringToTest	:= "hello",
			EqualToString	:= 'hello',
			EqualToWString	:= "hello",
			IgnoreCases		:= FALSE,
			ExpectedResult	:= FALSE,
			typeToTest		:= TypeToTest.TEST_STRING ),

		// test number 11
		( 	StringToTest	:= 'Давным-давно, когда тигр курил',
			WStringToTest	:= "Давным-давно, когда тигр курил",
			EqualToString	:= 'Давным-давно, когда тигр курил',
			EqualToWString	:= "Давным-давно, когда тигр курил",
			IgnoreCases		:= FALSE,
			ExpectedResult	:= FALSE,
			typeToTest		:= TypeToTest.TEST_STRING ),
			
		// test number 12
		( 	StringToTest	:= 'לאנג צוריק ווען טיגערס פלעגן רייכערן',
			WStringToTest	:= "לאנג צוריק ווען טיגערס פלעגן רייכערן",
			EqualToString	:= 'לאנג צוריק ווען טיגערס פלעגן רייכערן',
			EqualToWString	:= "לאנג צוריק ווען טיגערס פלעגן רייכערן",
			IgnoreCases		:= FALSE,
			ExpectedResult	:= FALSE,
			typeToTest		:= TypeToTest.TEST_STRING ),
			
		// test number 13
		( 	StringToTest	:= 'Давным-давно, когда тигркурил',
			WStringToTest	:= "Давным-давно, когда тигркурил",
			EqualToString	:= 'Давным-давно, когда тигр курил',
			EqualToWString	:= "Давным-давно, когда тигр курил",
			IgnoreCases		:= FALSE,
			ExpectedResult	:= TRUE,
			typeToTest		:= TypeToTest.TEST_STRING ),
			
		// test number 14
		( 	StringToTest	:= 'לאנג צוריק ווען טיגערס פלעגןרייכערן',
			WStringToTest	:= "לאנג צוריק ווען טיגערס פלעגןרייכערן",
			EqualToString	:= 'לאנג צוריק ווען טיגערס פלעגן רייכערן',
			EqualToWString	:= "לאנג צוריק ווען טיגערס פלעגן רייכערן",
			IgnoreCases		:= FALSE,
			ExpectedResult	:= TRUE,
			typeToTest		:= TypeToTest.TEST_STRING ),
			
		// test number 15
		( 	StringToTest	:= 'לאנג צוריק ווען טיגערס פלעגןרייכערן',
			WStringToTest	:= "לאנג צוריק ווען טיגערס פלעגןרייכערן",
			EqualToString	:= 'לאנג צוריק ווע טיגערס פלעגןרייכערן',
			EqualToWString	:= "לאנג צוריק ווע טיגערס פלעגןרייכערן",
			IgnoreCases		:= FALSE,
			ExpectedResult	:= TRUE,
			typeToTest		:= TypeToTest.TEST_STRING ),
			
		// test number 16
		( 	StringToTest	:= '',
			WStringToTest	:= "",
			EqualToString	:= '',
			EqualToWString	:= "",
			IgnoreCases		:= FALSE,
			ExpectedResult	:= FALSE,
			typeToTest		:= TypeToTest.TEST_STRING ),
			
		// test number 17
		( 	StringToTest	:= ' ',
			WStringToTest	:= " ",
			EqualToString	:= '  ',
			EqualToWString	:= "  ",
			IgnoreCases		:= FALSE,
			ExpectedResult	:= TRUE,
			typeToTest		:= TypeToTest.TEST_STRING ),
			
		// test number 18
		( 	StringToTest	:= 'abc',
			WStringToTest	:= "abc",
			EqualToString	:= 'ABC',
			EqualToWString	:= "ABC",
			IgnoreCases		:= TRUE,
			ExpectedResult	:= FALSE,
			typeToTest		:= TypeToTest.TEST_STRING ),

		// test number 19
		( 	StringToTest	:= 'нефти и газа',
			WStringToTest	:= "нефти и газа",
			EqualToString	:= 'НЕФТИ И ГАЗА',
			EqualToWString	:= "НЕФТИ И ГАЗА",
			IgnoreCases		:= TRUE,
			ExpectedResult	:= FALSE,
			typeToTest		:= TypeToTest.TEST_STRING ),
			
		// test number 20
		( 	StringToTest	:= 'нефти и газа',
			WStringToTest	:= "нефти и газа",
			EqualToString	:= 'НЕФТИ И ГАЗА',
			EqualToWString	:= "НЕФТИ И ГАЗА",
			IgnoreCases		:= TRUE,
			ExpectedResult	:= FALSE,
			typeToTest		:= TypeToTest.TEST_STRING ),

		// test number 21
		( 	StringToTest	:= '',
			WStringToTest	:= "🧐",
			EqualToString	:= '',
			EqualToWString	:= "🧐",
			IgnoreCases		:= TRUE,
			ExpectedResult	:= FALSE,
			typeToTest		:= TypeToTest.TEST_WSTRING ),
			
		// test number 22
		( 	StringToTest	:= '',
			WStringToTest	:= "🧐",
			EqualToString	:= '',
			EqualToWString	:= "🧐",
			IgnoreCases		:= FALSE,
			ExpectedResult	:= FALSE,
			typeToTest		:= TypeToTest.TEST_WSTRING ),
			
		// test number 23
		( 	StringToTest	:= '',
			WStringToTest	:= "h🧐",
			EqualToString	:= '',
			EqualToWString	:= "h🧐",
			IgnoreCases		:= TRUE,
			ExpectedResult	:= FALSE,
			typeToTest		:= TypeToTest.TEST_WSTRING ),
			
		// test number 24
		( 	StringToTest	:= '',
			WStringToTest	:= "h🧐",
			EqualToString	:= '',
			EqualToWString	:= "h🧐",
			IgnoreCases		:= FALSE,
			ExpectedResult	:= FALSE,
			typeToTest		:= TypeToTest.TEST_WSTRING ),
			
		// test number 25
		( 	StringToTest	:= '',
			WStringToTest	:= "h🧐",
			EqualToString	:= '',
			EqualToWString	:= "h🧐 ",
			IgnoreCases		:= TRUE,
			ExpectedResult	:= TRUE,
			typeToTest		:= TypeToTest.TEST_WSTRING ),
			
		// test number 26
		( 	StringToTest	:= '',
			WStringToTest	:= "h🧐",
			EqualToString	:= '',
			EqualToWString	:= "h🧐 ",
			IgnoreCases		:= FALSE,
			ExpectedResult	:= TRUE,
			typeToTest		:= TypeToTest.TEST_WSTRING ),
			
		// test number 27
		( 	StringToTest	:= '$$00434',
			WStringToTest	:= "$$00434",
			EqualToString	:= '$$00434',
			EqualToWString	:= "$$00434",
			IgnoreCases		:= FALSE,
			ExpectedResult	:= FALSE,
			typeToTest		:= TypeToTest.TEST_WSTRING ),
			
		// test number 28
		( 	StringToTest	:= '$$00434',
			WStringToTest	:= "$$00434",
			EqualToString	:= '$$00434',
			EqualToWString	:= "$$00434",
			IgnoreCases		:= TRUE,
			ExpectedResult	:= FALSE,
			typeToTest		:= TypeToTest.TEST_WSTRING ),
			
		// test number 29
		( 	StringToTest	:= '$$00434',
			WStringToTest	:= "$$00434",
			EqualToString	:= '$$00434',
			EqualToWString	:= "$$00434",
			IgnoreCases		:= FALSE,
			ExpectedResult	:= FALSE,
			typeToTest		:= TypeToTest.TEST_STRING ),
			
		// test number 30
		( 	StringToTest	:= '$$00434',
			WStringToTest	:= "$$00434",
			EqualToString	:= '$$00434',
			EqualToWString	:= "$$00434",
			IgnoreCases		:= TRUE,
			ExpectedResult	:= FALSE,
			typeToTest		:= TypeToTest.TEST_STRING ),
			
		// test number 31
		( 	StringToTest	:= '2',
			WStringToTest	:= "2",
			EqualToString	:= '²',
			EqualToWString	:= "²",
			IgnoreCases		:= TRUE,
			ExpectedResult	:= TRUE,
			typeToTest		:= TypeToTest.TEST_STRING ),
			
		// test number 32
		( 	StringToTest	:= '2',
			WStringToTest	:= "2",
			EqualToString	:= '²',
			EqualToWString	:= "²",
			IgnoreCases		:= TRUE,
			ExpectedResult	:= TRUE,
			typeToTest		:= TypeToTest.TEST_WSTRING )
						
	];
END_VAR

// ---- AssertionTester/AssertionTests/StringAssertions/TestDataSets/IsLengthBetweenDataSet.TcGVL
(*

short summary
=============

.. <legal notes>

legal notes
=================
| SPDX-FileCopyrightText: © 2023 ekvip automation GmbH <info@ekvip.de>
| SPDX-License-Identifier: Apache-2.0
| For details check: Apache-2.0_

.. _Apache-2.0: https://www.apache.org/licenses/LICENSE-2.0

.. </legal notes>

*)

{warning 'header is generated please add your documentation'}
{attribute 'qualified_only'}
VAR_GLOBAL CONSTANT
	SIZE_OF_LENGTHBETWEEN_DATASET:USINT := 18;
END_VAR

VAR_GLOBAL
	isLenghtBetweenToDataSetCommon : ARRAY[0..SIZE_OF_LENGTHBETWEEN_DATASET] OF IsLengthBetweenBasicData := [
		// test number 0
		( 	StringToTest	:= 'hello',
			WStringToTest	:= "hello",
			ExpectedResult 	:= FALSE,
			maxLength		:= 9,
			minLength		:= 3,
			typeToTest      :=  TypeToTest.TEST_WSTRING   )	,

		// test number 1
		( 	StringToTest	:= 'привет',
			WStringToTest	:= "привет",
			ExpectedResult 	:= FALSE,
			maxLength		:= 9,
			minLength		:= 3,
			typeToTest      :=  TypeToTest.TEST_WSTRING   ),	

		// test number 2
		( 	StringToTest	:= 'hello',
			WStringToTest	:= "hello",
			ExpectedResult 	:= FALSE,
			maxLength		:= 9,
			minLength		:= 3,
			typeToTest      :=  TypeToTest.TEST_STRING   ),

		// test number 3
		( 	StringToTest	:= 'привет',
			WStringToTest	:= "привет",
			ExpectedResult 	:= FALSE,
			maxLength		:= 9,
			minLength		:= 3,
			typeToTest      :=  TypeToTest.TEST_STRING   ),

		// test number 4
		( 	StringToTest	:= '',
			WStringToTest	:= "",
			ExpectedResult 	:= FALSE,
			maxLength		:= 1,
			minLength		:= 0,
			typeToTest      :=  TypeToTest.TEST_STRING   ),
			
		// test number 5
		( 	StringToTest	:= '   ',
			WStringToTest	:= "   ",
			ExpectedResult 	:= FALSE,
			maxLength		:= 4,
			minLength		:= 0,
			typeToTest      :=  TypeToTest.TEST_STRING   ),
			
		// test number 6
		( 	StringToTest	:= 'computer',
			WStringToTest	:= "computer",
			ExpectedResult 	:= TRUE,
			maxLength		:= 4,
			minLength		:= 0,
			typeToTest      :=  TypeToTest.TEST_STRING   ),
			
		// test number 7
		( 	StringToTest	:= 'העלא',
			WStringToTest	:= "העלא",
			ExpectedResult 	:= TRUE,
			maxLength		:= 2,
			minLength		:= 0,
			typeToTest      :=  TypeToTest.TEST_STRING   ),

		// test number 8
		( 	StringToTest	:= '',
			WStringToTest	:= "",
			ExpectedResult 	:= FALSE,
			maxLength		:= 1,
			minLength		:= 0,
			typeToTest      :=  TypeToTest.TEST_WSTRING   ),
			
		// test number 9
		( 	StringToTest	:= '   ',
			WStringToTest	:= "   ",
			ExpectedResult 	:= FALSE,
			maxLength		:= 4,
			minLength		:= 0,
			typeToTest      :=  TypeToTest.TEST_WSTRING   ),
			
		// test number 10
		( 	StringToTest	:= 'computer',
			WStringToTest	:= "computer",
			ExpectedResult 	:= TRUE,
			maxLength		:= 4,
			minLength		:= 0,
			typeToTest      :=  TypeToTest.TEST_WSTRING   ),
			
		// test number 11
		( 	StringToTest	:= 'העלא',
			WStringToTest	:= "העלא",
			ExpectedResult 	:= TRUE,
			maxLength		:= 2,
			minLength		:= 0,
			typeToTest      :=  TypeToTest.TEST_WSTRING   ),
			
		// test number 12
		( 	StringToTest	:= 'העלא',
			WStringToTest	:= "העלא",
			ExpectedResult 	:= TRUE,
			maxLength		:= 2,
			minLength		:= 0,
			typeToTest      :=  TypeToTest.TEST_WSTRING   ),

		// test number 13
		( 	StringToTest	:= 'העלא asdsda  sadad',
			WStringToTest	:= "העלא asdsda  sadad",
			ExpectedResult 	:= FALSE,
			maxLength		:= 20,
			minLength		:= 10,
			typeToTest      :=  TypeToTest.TEST_WSTRING   ),

		// test number 14
		( 	StringToTest	:= 'העלא asdsda  sadad',
			WStringToTest	:= "העלא asdsda  sadad",
			ExpectedResult 	:= FALSE,
			maxLength		:= 20,
			minLength		:= 10,
			typeToTest      :=  TypeToTest.TEST_STRING   ),

		// test number 15
		( 	StringToTest	:= '',
			WStringToTest	:= "👩‍🔧",
			ExpectedResult 	:= FALSE,
			maxLength		:= 10,
			minLength		:= 0,
			typeToTest      :=  TypeToTest.TEST_WSTRING   ),

		// test number 16
		( 	StringToTest	:= '',
			WStringToTest	:= "👩‍🔧",
			ExpectedResult 	:= TRUE,
			maxLength		:= 2,
			minLength		:= 0,
			typeToTest      :=  TypeToTest.TEST_WSTRING   ),

		// test number 17
		( 	StringToTest	:= '595',
			WStringToTest	:= "595",
			ExpectedResult 	:= FALSE,
			maxLength		:= 5,
			minLength		:= 2,
			typeToTest      :=  TypeToTest.TEST_WSTRING  ),	

		// test number 18
		( 	StringToTest	:= '595',
			WStringToTest	:= "595",
			ExpectedResult 	:= FALSE,
			maxLength		:= 5,
			minLength		:= 2,
			typeToTest      :=  TypeToTest.TEST_STRING  )

		
			
	];
END_VAR

// ---- AssertionTester/AssertionTests/StringAssertions/TestDataSets/IsLengthTestDataSet.TcGVL
(*

short summary
=============

.. <legal notes>

legal notes
=================
| SPDX-FileCopyrightText: © 2023 ekvip automation GmbH <info@ekvip.de>
| SPDX-License-Identifier: Apache-2.0
| For details check: Apache-2.0_

.. _Apache-2.0: https://www.apache.org/licenses/LICENSE-2.0

.. </legal notes>

*)

{warning 'header is generated please add your documentation'}
{attribute 'qualified_only'}
VAR_GLOBAL CONSTANT
	SIZE_OF_IS_DATASET:USINT := 61;
END_VAR

VAR_GLOBAL
	IsLenghtDataSetCommon : ARRAY[0..SIZE_OF_IS_DATASET] OF IsLengthBasicData := [

	// test number 0 
	  (	StringToTest	:= '',     	
		ExpectedResult	:= FALSE, 
		ExpectedLength 	:= 0,   
		funcType 		:= FunctionType.EXACT, 	
		typeToTest		:= TypeToTest.TEST_STRING),

	// test number 1 		
   	 (	StringToTest	:= 'abgf', 	
		ExpectedResult	:= FALSE, 
		ExpectedLength 	:= 4 , 
		funcType 		:= FunctionType.EXACT, 	
		typeToTest		:= TypeToTest.TEST_STRING),
		
	// test number 2		
	  ( StringToTest	:= '    ', 	
		ExpectedResult	:= FALSE, 
		ExpectedLength 	:= 4 , 
		funcType 		:= FunctionType.EXACT, 	
		typeToTest		:= TypeToTest.TEST_STRING),
		
	// test number 3			
	  ( StringToTest	:= '',     	
		ExpectedResult	:= TRUE,  
		ExpectedLength 	:= 3,   
		funcType 		:= FunctionType.EXACT,	
		typeToTest		:= TypeToTest.TEST_STRING),
		
	// test number 4	   			
	  ( StringToTest	:= 'abgf', 	
		ExpectedResult	:= TRUE,  
		ExpectedLength 	:= 6 , 
		funcType 		:= FunctionType.EXACT,  	
		typeToTest		:= TypeToTest.TEST_STRING),
		
	// test number 5			
	  ( StringToTest	:= '    ', 	
		ExpectedResult	:= TRUE,  
		ExpectedLength 	:= 6 , 
		funcType 		:= FunctionType.EXACT,  	
		typeToTest		:= TypeToTest.TEST_STRING),
		
	// test number 6		  
	  ( StringToTest	:= '%/&)(/)//',
		ExpectedResult	:= FALSE, 
		ExpectedLength 	:= 9, 
		funcType		:= FunctionType.EXACT,  
		typeToTest		:= TypeToTest.TEST_STRING),

	// test number 7		  
	  (  					   	
		ExpectedResult	:= FALSE , 
		ExpectedLength 	:= 0, 
		funcType		:= FunctionType.EXACT,  
		typeToTest		:= TypeToTest.TEST_STRING),
	
	// test number 8
	  ( StringToTest	:= '',     
		ExpectedResult	:= FALSE, 
		ExpectedLength 	:= 0,   
		funcType		:= FunctionType.MAXIMUM, 	
 		typeToTest		:= TypeToTest.TEST_STRING),

	// test number 9   			
	  ( StringToTest	:= 'abgf', 
		ExpectedResult	:= FALSE, 
		ExpectedLength 	:= 4, 
		funcType		:= FunctionType.MAXIMUM, 	
		typeToTest		:= TypeToTest.TEST_STRING),

	// test number 10		
	  ( StringToTest	:= '    ', 
		ExpectedResult	:= FALSE, 
		ExpectedLength 	:= 4 , 
		funcType		:= FunctionType.MAXIMUM, 	
		typeToTest		:= TypeToTest.TEST_STRING),

	// test number 11		
	  ( StringToTest	:= '',     
		ExpectedResult	:= FALSE, 
		ExpectedLength 	:= 8,   
		funcType		:= FunctionType.MAXIMUM,	
		typeToTest		:= TypeToTest.TEST_STRING),

	// test number 12   			
	  ( StringToTest	:= 'abgf', 
		ExpectedResult	:= FALSE, 
		ExpectedLength 	:= 6, 
		funcType		:= FunctionType.MAXIMUM,  
		typeToTest		:= TypeToTest.TEST_STRING),

	// test number 13		
	  ( StringToTest	:= '    ', 
		ExpectedResult	:= FALSE, 
		ExpectedLength 	:= 6, 
		funcType		:= FunctionType.MAXIMUM,  
		typeToTest		:= TypeToTest.TEST_STRING),

	// test number 14		
	  ( ExpectedResult	:= FALSE , 
		ExpectedLength 	:= 0 , 
		funcType		:= FunctionType.MAXIMUM,  
		typeToTest		:= TypeToTest.TEST_STRING),

	// test number 15
	  ( StringToTest	:= '', 
		ExpectedResult	:= FALSE, 
		ExpectedLength 	:= 0, 
		funcType		:= FunctionType.MINIMUM,  
		typeToTest		:= TypeToTest.TEST_STRING),

	// test number 16	  
	  ( StringToTest	:= 'hello', 
		ExpectedResult	:= FALSE, 
		ExpectedLength 	:= 5, 
		funcType		:= FunctionType.MINIMUM,  
		typeToTest		:= TypeToTest.TEST_STRING),

	// test number 17	
	  ( StringToTest	:= 'привет', 
		ExpectedResult	:= FALSE, 
		ExpectedLength 	:= 5, 
		funcType		:= FunctionType.MINIMUM,  
		typeToTest		:= TypeToTest.TEST_STRING),

	// test number 18
	  ( StringToTest	:= '', 
		ExpectedResult	:= TRUE, 
		ExpectedLength 	:= 4, 
		funcType		:= FunctionType.MINIMUM,  
		typeToTest		:= TypeToTest.TEST_STRING),
	  
	// test number 19	
	  ( StringToTest	:= 'hello', 
		ExpectedResult	:= TRUE, 
		ExpectedLength 	:= 7, 
		funcType		:= FunctionType.MINIMUM,  
		typeToTest		:= TypeToTest.TEST_STRING),

	// test number 20	
	  ( StringToTest	:= 'привет', 
		ExpectedResult	:= TRUE, 
		ExpectedLength 	:= 10, 
		funcType		:= FunctionType.MINIMUM,  
		typeToTest		:= TypeToTest.TEST_STRING),

	// test number 21	
	  ( StringToTest	:= '    ', 
		ExpectedResult	:= FALSE, 
		ExpectedLength 	:= 4, 
		funcType		:= FunctionType.MINIMUM,  
		typeToTest		:= TypeToTest.TEST_STRING),
	
	// test number 22	
	  ( StringToTest	:= '    ', 
		ExpectedResult	:= TRUE, 
		ExpectedLength 	:= 5, 
		funcType		:= FunctionType.MINIMUM,  
		typeToTest		:= TypeToTest.TEST_STRING),

	// test number 23	
	  ( StringToTest	:= '    ', 
		ExpectedResult	:= TRUE, 
		ExpectedLength 	:= 10, 
		funcType		:= FunctionType.MINIMUM,  
		typeToTest		:= TypeToTest.TEST_STRING),
		
	// test number 24	
	  ( StringToTest	:= '%/&)(/)//',
		ExpectedResult	:= FALSE, 
		ExpectedLength 	:= 9, 
		funcType		:= FunctionType.MINIMUM,  
		typeToTest		:= TypeToTest.TEST_STRING),
		
	// test number 25	
	  ( StringToTest	:= '%/&)(/)//',
		ExpectedResult	:= TRUE, 
		ExpectedLength 	:= 10, 
		funcType		:= FunctionType.MINIMUM,  
		typeToTest		:= TypeToTest.TEST_STRING),

	// test number 26	
	  ( WStringToTest	:= "", 			
		ExpectedResult	:= FALSE,	
		ExpectedLength 	:= 0, 	
		funcType		:= FunctionType.EXACT, 
		typeToTest		:= TypeToTest.TEST_WSTRING),

	// test number 27		
	  ( WStringToTest	:= "abc" , 			
		ExpectedResult	:= FALSE, 
		ExpectedLength 	:= 3 , 	
		funcType		:= FunctionType.EXACT ,	
		typeToTest		:= TypeToTest.TEST_WSTRING),

	// test number 28		
	  ( WStringToTest	:= "хороший", 		
		ExpectedResult	:= FALSE, 
		ExpectedLength 	:= 7, 	
		funcType		:= FunctionType.EXACT , 
		typeToTest		:= TypeToTest.TEST_WSTRING),

	// test number 29		
	  ( WStringToTest	:= "хороший abc", 	
		ExpectedResult	:= FALSE, 
		ExpectedLength 	:= 11, 	
		funcType		:= FunctionType.EXACT , 
		typeToTest		:= TypeToTest.TEST_WSTRING),

	// test number 30		
	  ( WStringToTest	:= "", 			
		ExpectedResult	:= TRUE, 	
		ExpectedLength 	:= 2, 	
		funcType		:= FunctionType.EXACT , 
		typeToTest		:= TypeToTest.TEST_WSTRING),
		
	// test number 31		
	  ( WStringToTest	:= "abc", 			
		ExpectedResult	:= TRUE, 	
		ExpectedLength 	:= 2,  	
		funcType		:= FunctionType.EXACT , 
		typeToTest		:= TypeToTest.TEST_WSTRING),
		
	// test number 32		
	  ( WStringToTest	:= "хороший", 		
		ExpectedResult	:= TRUE, 	
		ExpectedLength	:= 2, 	
		funcType		:= FunctionType.EXACT, 	
		typeToTest		:= TypeToTest.TEST_WSTRING),

	// test number 33		
	  ( WStringToTest	:= "хороший abc", 	
		ExpectedResult	:= TRUE, 	
		ExpectedLength 	:= 10, 	
		funcType		:= FunctionType.EXACT, 	
		typeToTest		:= TypeToTest.TEST_WSTRING),
		
	// test number 34		
	  ( WStringToTest	:= "    ", 		
		ExpectedResult	:= FALSE, 
		ExpectedLength 	:= 4, 	
		funcType		:= FunctionType.EXACT, 	
		typeToTest		:= TypeToTest.TEST_WSTRING),

	// test number 35		
	  ( WStringToTest	:= "صباح الخي", 	
		ExpectedResult	:= FALSE, 
		ExpectedLength 	:= 9,  	
		funcType		:= FunctionType.EXACT, 	
		typeToTest		:= TypeToTest.TEST_WSTRING),

	// test number 36		
	  ( WStringToTest	:= "😀", 			
		ExpectedResult	:= FALSE, 
		ExpectedLength 	:= 1,  	
		funcType		:= FunctionType.EXACT, 	
		typeToTest		:= TypeToTest.TEST_WSTRING),

	// test number 37		
	  ( WStringToTest	:= "%/&)(/)//", 	
		ExpectedResult	:= FALSE,
		ExpectedLength 	:= 9, 
		funcType		:= FunctionType.EXACT,  	
		typeToTest		:= TypeToTest.TEST_WSTRING),

	// test number 38		
	  ( ExpectedResult	:= FALSE ,
		ExpectedLength 	:= 0 , 
		funcType		:= FunctionType.EXACT,  	
		typeToTest		:= TypeToTest.TEST_WSTRING),

	// test number 39	
	  ( WStringToTest	:= "", 			
		ExpectedResult	:= FALSE,	
		ExpectedLength 	:= 0, 	
		funcType		:= FunctionType.MAXIMUM, 	
		typeToTest		:= TypeToTest.TEST_WSTRING),
		
	// test number 40		
	  ( WStringToTest	:= "abc", 			
		ExpectedResult	:= FALSE, 
		ExpectedLength	:= 3 , 	
       	funcType		:= FunctionType.MAXIMUM ,	
		typeToTest		:= TypeToTest.TEST_WSTRING),
		
	// test number 41		
	  ( WStringToTest	:= "хороший" , 		
		ExpectedResult	:= FALSE, 
		ExpectedLength 	:= 7, 	
		funcType		:= FunctionType.MAXIMUM , 	
		typeToTest		:= TypeToTest.TEST_WSTRING),
		
	// test number 42		
	  ( WStringToTest	:= "хороший abc", 	
		ExpectedResult	:= FALSE, 
		ExpectedLength 	:= 11, 	
		funcType		:= FunctionType.MAXIMUM ,	
		typeToTest		:= TypeToTest.TEST_WSTRING),
		
	// test number 43		
	  ( WStringToTest	:= "" , 			
		ExpectedResult	:= FALSE, 
		ExpectedLength 	:= 2, 	
		funcType		:= FunctionType.MAXIMUM ,
		typeToTest		:= TypeToTest.TEST_WSTRING),
		
	// test number 44		
	  ( WStringToTest	:= "abc" , 			
		ExpectedResult	:= TRUE,  
		ExpectedLength 	:= 2,  	
		funcType		:= FunctionType.MAXIMUM , 	
		typeToTest		:= TypeToTest.TEST_WSTRING),
		
	// test number 45		
	  ( WStringToTest	:= "хороший" , 		
		ExpectedResult	:= TRUE,  
		ExpectedLength 	:= 2, 	
		funcType		:= FunctionType.MAXIMUM, 	
		typeToTest		:= TypeToTest.TEST_WSTRING),
		
	// test number 46		
	  ( WStringToTest	:= "хороший abc" , 	
		ExpectedResult	:= FALSE, 
		ExpectedLength 	:= 18 , 	
		funcType		:= FunctionType.MAXIMUM, 	
		typeToTest		:= TypeToTest.TEST_WSTRING),
		
	// test number 47		
	  ( WStringToTest 	:= "    ", 		
		ExpectedResult	:= FALSE,  
		ExpectedLength 	:= 4 , 	
		funcType		:= FunctionType.MAXIMUM, 	
		typeToTest		:= TypeToTest.TEST_WSTRING),
		
	// test number 48		
	  ( WStringToTest	:= "صباح الخي" , 	
		ExpectedResult	:= FALSE, 
		ExpectedLength 	:= 9 ,  	
		funcType		:= FunctionType.MAXIMUM, 	
		typeToTest		:= TypeToTest.TEST_WSTRING),
		
	// test number 49		
	  ( WStringToTest	:= "😀" , 			
		ExpectedResult	:= FALSE, 
		ExpectedLength 	:= 9 ,  	
		funcType		:= FunctionType.MAXIMUM, 	
		typeToTest		:= TypeToTest.TEST_WSTRING),
		
	// test number 50		
	  ( ExpectedResult	:= FALSE, 
		ExpectedLength 	:= 0 , 	
		funcType		:= FunctionType.MAXIMUM,	
		typeToTest		:= TypeToTest.TEST_WSTRING),

	// test number 51
	  ( WStringToTest	:= "", 
		ExpectedResult	:= FALSE, 
		ExpectedLength 	:= 0, 
		funcType		:= FunctionType.MINIMUM,  
		typeToTest		:= TypeToTest.TEST_WSTRING),

	// test number 52	  
	  ( WStringToTest	:= "hello", 
		ExpectedResult	:= FALSE, 
		ExpectedLength 	:= 5, 
		funcType		:= FunctionType.MINIMUM,  
		typeToTest		:= TypeToTest.TEST_WSTRING),

	// test number 53	
	  ( WStringToTest	:= "привет", 
		ExpectedResult	:= FALSE, 
		ExpectedLength 	:= 5, 
		funcType		:= FunctionType.MINIMUM,  
		typeToTest		:= TypeToTest.TEST_WSTRING),

	// test number 54
	  ( WStringToTest	:= "", 
		ExpectedResult	:= TRUE, 
		ExpectedLength 	:= 4, 
		funcType		:= FunctionType.MINIMUM,  
		typeToTest		:= TypeToTest.TEST_WSTRING),
	  
	// test number 55	
	  ( WStringToTest	:= "hello", 
		ExpectedResult	:= TRUE, 
		ExpectedLength 	:= 7, 
		funcType		:= FunctionType.MINIMUM,  
		typeToTest		:= TypeToTest.TEST_WSTRING),

	// test number 56	
	  ( WStringToTest	:= "привет", 
		ExpectedResult	:= TRUE, 
		ExpectedLength 	:= 10, 
		funcType		:= FunctionType.MINIMUM,  
		typeToTest		:= TypeToTest.TEST_WSTRING),

	// test number 57	
	  ( WStringToTest	:= "    ", 
		ExpectedResult	:= FALSE, 
		ExpectedLength 	:= 4, 
		funcType		:= FunctionType.MINIMUM,  
		typeToTest		:= TypeToTest.TEST_WSTRING),
	
	// test number 58	
	  ( WStringToTest	:= "    ", 
		ExpectedResult	:= TRUE, 
		ExpectedLength 	:= 5, 
		funcType		:= FunctionType.MINIMUM,  
		typeToTest		:= TypeToTest.TEST_WSTRING),

	// test number 59	
	  ( WStringToTest	:= "    ", 
		ExpectedResult	:= TRUE, 
		ExpectedLength 	:= 10, 
		funcType		:= FunctionType.MINIMUM,  
		typeToTest		:= TypeToTest.TEST_WSTRING),
		
	// test number 60	
	  ( WStringToTest	:= "%/&)(/)//",
		ExpectedResult	:= FALSE, 
		ExpectedLength 	:= 9, 
		funcType		:= FunctionType.MINIMUM,  
		typeToTest		:= TypeToTest.TEST_WSTRING),
		
	// test number 61	
	  ( WStringToTest	:= "%/&)(/)//",
		ExpectedResult	:= TRUE, 
		ExpectedLength 	:= 10, 
		funcType		:= FunctionType.MINIMUM,  
		typeToTest		:= TypeToTest.TEST_WSTRING)

	
];
END_VAR

// ---- AssertionTester/AssertionTests/StringAssertions/TestDataSets/isNotEmtyTestDataSet.TcGVL
(*

short summary
=============

.. <legal notes>

legal notes
=================
| SPDX-FileCopyrightText: © 2023 ekvip automation GmbH <info@ekvip.de>
| SPDX-License-Identifier: Apache-2.0
| For details check: Apache-2.0_

.. _Apache-2.0: https://www.apache.org/licenses/LICENSE-2.0

.. </legal notes>

*)

{warning 'header is generated please add your documentation'}
{attribute 'qualified_only'}
VAR_GLOBAL CONSTANT
	SIZE_OF_ISNOTEMPTY_DATASET:USINT := 13;
END_VAR

VAR_GLOBAL
	isNotEmptyDataSetCommon : ARRAY[0..SIZE_OF_ISNOTEMPTY_DATASET] OF isEmptyDataStr := [
		// test number 0
		(	StringToTest 	:= 'hello',
			WStringToTest 	:= "hello",
			ExpectedResult  := FALSE,
			typeToTest     	:= TypeToTest.TEST_STRING ),
		
		// test number 1
		(	StringToTest 	:= 'hello',
			WStringToTest 	:= "hello",
			ExpectedResult  := FALSE,
			typeToTest     	:= TypeToTest.TEST_STRING ),

		// test number 2
		(	StringToTest 	:= '',
			WStringToTest 	:= "",
			ExpectedResult  := TRUE,
			typeToTest     	:= TypeToTest.TEST_STRING ),		
		
		// test number 3
		(	StringToTest 	:= '',
			WStringToTest 	:= "",
			ExpectedResult  := TRUE,
			typeToTest     	:= TypeToTest.TEST_WSTRING ),	

		// test number 4
		(	StringToTest 	:= '   ',
			WStringToTest 	:= "   ",
			ExpectedResult  := FALSE,
			typeToTest     	:= TypeToTest.TEST_WSTRING ),

		// test number 5
		(	StringToTest 	:= '   ',
			WStringToTest 	:= "   ",
			ExpectedResult  := FALSE,
			typeToTest     	:= TypeToTest.TEST_STRING ),
			
		// test number 6
		(	StringToTest 	:= '   ',
			WStringToTest 	:= "नमस्ते",
			ExpectedResult  := FALSE,
			typeToTest     	:= TypeToTest.TEST_WSTRING ),
				
		// test number 7
		(	StringToTest 	:= 'мальчик или девочка',
			WStringToTest 	:= "мальчик или девочка",
			ExpectedResult  := FALSE,
			typeToTest     	:= TypeToTest.TEST_WSTRING ),
			
		// test number 8
		(	StringToTest 	:= 'мальчик или девочка',
			WStringToTest 	:= "мальчик или девочка",
			ExpectedResult  := FALSE,
			typeToTest     	:= TypeToTest.TEST_STRING ),
			
		// test number 9
		(	StringToTest 	:= '',
			WStringToTest 	:= "👨‍🔬 👩‍🎨 🧑‍🎨 👨‍🎨 👩‍🚒 🧑‍🚒 👨‍🚒 👩‍✈️ 🧑‍✈️ 👨‍✈️ 👩‍🚀",
			ExpectedResult  := FALSE,
			typeToTest     	:= TypeToTest.TEST_WSTRING ),
			
		// test number 10
		(	StringToTest 	:= 'QQQqqqq@@@@@%%%%',
			WStringToTest 	:= "QQQqqqq@@@@@%%%%",
			ExpectedResult  := FALSE,
			typeToTest     	:= TypeToTest.TEST_WSTRING ),

		// test number 11
		(	StringToTest 	:= '.',
			WStringToTest 	:= ".",
			ExpectedResult  := FALSE,
			typeToTest     	:= TypeToTest.TEST_WSTRING ),

		// test number 12
		(	StringToTest 	:= 'QQQqqqq@@@@@%%%%',
			WStringToTest 	:= "QQQqqqq@@@@@%%%%",
			ExpectedResult  := FALSE,
			typeToTest     	:= TypeToTest.TEST_STRING ),

		// test number 13
		(	StringToTest 	:= '.',
			WStringToTest 	:= ".",
			ExpectedResult  := FALSE,
			typeToTest     	:= TypeToTest.TEST_STRING )		


	];
END_VAR

// ---- AssertionTester/AssertionTests/StringAssertions/TestDataSets/isNotEqualToTestDataSet.TcGVL
(*

short summary
=============

.. <legal notes>

legal notes
=================
| SPDX-FileCopyrightText: © 2023 ekvip automation GmbH <info@ekvip.de>
| SPDX-License-Identifier: Apache-2.0
| For details check: Apache-2.0_

.. _Apache-2.0: https://www.apache.org/licenses/LICENSE-2.0

.. </legal notes>

*)

{warning 'header is generated please add your documentation'}
{attribute 'qualified_only'}
VAR_GLOBAL CONSTANT
	SIZE_OF_ISNOTEQUALTO_DATASET:USINT := 27;
END_VAR

VAR_GLOBAL
	isNotEqualDataSetCommon : ARRAY[0..SIZE_OF_ISNOTEQUALTO_DATASET] OF isEqualToDataStr := [
		// test number 0
		( 	StringToTest	:= 'hello',
			WStringToTest	:= "hello",
			EqualToString	:= 'hello',
			EqualToWString	:= "hello",
			IgnoreCases		:= FALSE,
			ExpectedResult	:= TRUE,
			typeToTest		:= TypeToTest.TEST_WSTRING ),
			
		// test number 1
		( 	StringToTest	:= 'Давным-давно, когда тигр курил',
			WStringToTest	:= "Давным-давно, когда тигр курил",
			EqualToString	:= 'Давным-давно, когда тигр курил',
			EqualToWString	:= "Давным-давно, когда тигр курил",
			IgnoreCases		:= FALSE,
			ExpectedResult	:= TRUE,
			typeToTest		:= TypeToTest.TEST_WSTRING ),
			
		// test number 2
		( 	StringToTest	:= 'Давным-давно, когда тигр курил',
			WStringToTest	:= "Давным-давно, когда тигр курил",
			EqualToString	:= 'Давным-давно, когда тигр курил',
			EqualToWString	:= "Давным-давно, когда тигр курил",
			IgnoreCases		:= FALSE,
			ExpectedResult	:= TRUE,
			typeToTest		:= TypeToTest.TEST_STRING ),
			
		// test number 3
		( 	StringToTest	:= 'לאנג צוריק ווען טיגערס פלעגן רייכערן',
			WStringToTest	:= "לאנג צוריק ווען טיגערס פלעגן רייכערן",
			EqualToString	:= 'לאנג צוריק ווען טיגערס פלעגן רייכערן',
			EqualToWString	:= "לאנג צוריק ווען טיגערס פלעגן רייכערן",
			IgnoreCases		:= FALSE,
			ExpectedResult	:= TRUE,
			typeToTest		:= TypeToTest.TEST_WSTRING ),
			
		// test number 4
		( 	StringToTest	:= 'Давным-давно, когда тигркурил',
			WStringToTest	:= "Давным-давно, когда тигркурил",
			EqualToString	:= 'Давным-давно, когда тигр курил',
			EqualToWString	:= "Давным-давно, когда тигр курил",
			IgnoreCases		:= FALSE,
			ExpectedResult	:= FALSE,
			typeToTest		:= TypeToTest.TEST_WSTRING ),
			
		// test number 5
		( 	StringToTest	:= 'לאנג צוריק ווען טיגערס פלעגן רייכערן',
			WStringToTest	:= "לאנג צוריק ווען טיגערס פלעגן רייכערן",
			EqualToString	:= 'לאנג צוריק ווען טיגערס פלעגן רייכערן',
			EqualToWString	:= "לאנג צוריק ווען טיגערס פלעגן רייכערן",
			IgnoreCases		:= FALSE,
			ExpectedResult	:= TRUE,
			typeToTest		:= TypeToTest.TEST_STRING ),
			
		// test number 6
		( 	StringToTest	:= 'Давным-давно, когда тигркурил',
			WStringToTest	:= "Давным-давно, когда тигркурил",
			EqualToString	:= 'Давным-давно, когда тигр курил',
			EqualToWString	:= "Давным-давно, когда тигр курил",
			IgnoreCases		:= FALSE,
			ExpectedResult	:= False,
			typeToTest		:= TypeToTest.TEST_STRING ),

		// test number 7
		( 	StringToTest	:= '',
			WStringToTest	:= "",
			EqualToString	:= '',
			EqualToWString	:= "",
			IgnoreCases		:= FALSE,
			ExpectedResult	:= TRUE,
			typeToTest		:= TypeToTest.TEST_WSTRING ),
			
		// test number 8
		( 	StringToTest	:= ' ',
			WStringToTest	:= " ",
			EqualToString	:= '  ',
			EqualToWString	:= "  ",
			IgnoreCases		:= FALSE,
			ExpectedResult	:= FALSE,
			typeToTest		:= TypeToTest.TEST_WSTRING ),
			
		// test number 9
		( 	StringToTest	:= 'abc',
			WStringToTest	:= "abc",
			EqualToString	:= 'ABC',
			EqualToWString	:= "ABC",
			IgnoreCases		:= TRUE,
			ExpectedResult	:= TRUE,
			typeToTest		:= TypeToTest.TEST_WSTRING ),

		// test number 10
		( 	StringToTest	:= 'нефти и газа',
			WStringToTest	:= "нефти и газа",
			EqualToString	:= 'НЕФТИ И ГАЗА',
			EqualToWString	:= "НЕФТИ И ГАЗА",
			IgnoreCases		:= TRUE,
			ExpectedResult	:= TRUE,
			typeToTest		:= TypeToTest.TEST_WSTRING 	),	
        
		// test number 11
		( 	StringToTest	:= 'Давным-давно, когда тигркурил',
			WStringToTest	:= "Давным-давно, когда тигркурил",
			EqualToString	:= 'Давным-давно, когда тигр курил',
			EqualToWString	:= "Давным-давно, когда тигр курил",
			IgnoreCases		:= FALSE,
			ExpectedResult	:= False,
			typeToTest		:= TypeToTest.TEST_STRING ),

		// test number 12
		( 	StringToTest	:= '',
			WStringToTest	:= "",
			EqualToString	:= '',
			EqualToWString	:= "",
			IgnoreCases		:= FALSE,
			ExpectedResult	:= TRUE,
			typeToTest		:= TypeToTest.TEST_WSTRING ),
			
		// test number 13
		( 	StringToTest	:= ' ',
			WStringToTest	:= " ",
			EqualToString	:= '  ',
			EqualToWString	:= "  ",
			IgnoreCases		:= FALSE,
			ExpectedResult	:= FALSE,
			typeToTest		:= TypeToTest.TEST_WSTRING ),
			
		// test number 14
		( 	StringToTest	:= 'abc',
			WStringToTest	:= "abc",
			EqualToString	:= 'ABC',
			EqualToWString	:= "ABC",
			IgnoreCases		:= TRUE,
			ExpectedResult	:= TRUE,
			typeToTest		:= TypeToTest.TEST_WSTRING ),

		// test number 15
		( 	StringToTest	:= 'нефти и газа',
			WStringToTest	:= "нефти и газа",
			EqualToString	:= 'НЕФТИ И ГАЗА',
			EqualToWString	:= "НЕФТИ И ГАЗА",
			IgnoreCases		:= TRUE,
			ExpectedResult	:= TRUE,
			typeToTest		:= TypeToTest.TEST_WSTRING ),
			
		// test number 16
		( 	StringToTest	:= '',
			WStringToTest	:= "🧐",
			EqualToString	:= '',
			EqualToWString	:= "🧐",
			IgnoreCases		:= TRUE,
			ExpectedResult	:= TRUE,
			typeToTest		:= TypeToTest.TEST_WSTRING ),
			
		// test number 17
		( 	StringToTest	:= '',
			WStringToTest	:= "🧐",
			EqualToString	:= '',
			EqualToWString	:= "🧐",
			IgnoreCases		:= FALSE,
			ExpectedResult	:= TRUE,
			typeToTest		:= TypeToTest.TEST_WSTRING ),
			
		// test number 18
		( 	StringToTest	:= '',
			WStringToTest	:= "h🧐",
			EqualToString	:= '',
			EqualToWString	:= "h🧐",
			IgnoreCases		:= TRUE,
			ExpectedResult	:= TRUE,
			typeToTest		:= TypeToTest.TEST_WSTRING ),
			
		// test number 19
		( 	StringToTest	:= '',
			WStringToTest	:= "h🧐",
			EqualToString	:= '',
			EqualToWString	:= "h🧐",
			IgnoreCases		:= FALSE,
			ExpectedResult	:= TRUE,
			typeToTest		:= TypeToTest.TEST_WSTRING ),
			
		// test number 20
		( 	StringToTest	:= '',
			WStringToTest	:= "h🧐",
			EqualToString	:= '',
			EqualToWString	:= "h🧐 ",
			IgnoreCases		:= TRUE,
			ExpectedResult	:= FALSE,
			typeToTest		:= TypeToTest.TEST_WSTRING ),
			
		// test number 21
		( 	StringToTest	:= '',
			WStringToTest	:= "h🧐",
			EqualToString	:= '',
			EqualToWString	:= "h🧐 ",
			IgnoreCases		:= FALSE,
			ExpectedResult	:= FALSE,
			typeToTest		:= TypeToTest.TEST_WSTRING ),
			
		// test number 22
		( 	StringToTest	:= '$$00434',
			WStringToTest	:= "$$00434",
			EqualToString	:= '$$00434',
			EqualToWString	:= "$$00434",
			IgnoreCases		:= FALSE,
			ExpectedResult	:= TRUE,
			typeToTest		:= TypeToTest.TEST_WSTRING ),
			
		// test number 23
		( 	StringToTest	:= '$$00434',
			WStringToTest	:= "$$00434",
			EqualToString	:= '$$00434',
			EqualToWString	:= "$$00434",
			IgnoreCases		:= TRUE,
			ExpectedResult	:= TRUE,
			typeToTest		:= TypeToTest.TEST_WSTRING ),
			
		// test number 24
		( 	StringToTest	:= '$$00434',
			WStringToTest	:= "$$00434",
			EqualToString	:= '$$00434',
			EqualToWString	:= "$$00434",
			IgnoreCases		:= FALSE,
			ExpectedResult	:= TRUE,
			typeToTest		:= TypeToTest.TEST_STRING ),
			
		// test number 25
		( 	StringToTest	:= '$$00434',
			WStringToTest	:= "$$00434",
			EqualToString	:= '$$00434',
			EqualToWString	:= "$$00434",
			IgnoreCases		:= TRUE,
			ExpectedResult	:= TRUE,
			typeToTest		:= TypeToTest.TEST_STRING ),
			
		// test number 26
		( 	StringToTest	:= '2',
			WStringToTest	:= "2",
			EqualToString	:= '²',
			EqualToWString	:= "²",
			IgnoreCases		:= TRUE,
			ExpectedResult	:= FALSE,
			typeToTest		:= TypeToTest.TEST_STRING ),
			
		// test number 27
		( 	StringToTest	:= '2',
			WStringToTest	:= "2",
			EqualToString	:= '²',
			EqualToWString	:= "²",
			IgnoreCases		:= TRUE,
			ExpectedResult	:= FALSE,
			typeToTest		:= TypeToTest.TEST_WSTRING )
						
	];
END_VAR

// ---- AssertionTester/AssertionTests/StringAssertions/TestDataSets/startsWithDataSet.TcGVL
(*

short summary
=============

.. <legal notes>

legal notes
=================
| SPDX-FileCopyrightText: © 2023 ekvip automation GmbH <info@ekvip.de>
| SPDX-License-Identifier: Apache-2.0
| For details check: Apache-2.0_

.. _Apache-2.0: https://www.apache.org/licenses/LICENSE-2.0

.. </legal notes>

*)

{warning 'header is generated please add your documentation'}
{attribute 'qualified_only'}
VAR_GLOBAL CONSTANT
	SIZE_OF_STARTWITH_DATASET:USINT := 18 ;
END_VAR

VAR_GLOBAL
	StartsWithDataSetCommon : ARRAY[0..SIZE_OF_STARTWITH_DATASET] OF containsDataStr := [
		// Test number 0
		(	StringToTest		:= 'Hello',
		  	WStringToTest 		:= "Hello",
			StringToContain 	:= 'h',
			WStringToContain	:= "h",
			IgnoreCases			:= TRUE,
			Trim 				:= FALSE,
			ExpectedResult  	:= FALSE,
			typeToTest      	:= TypeToTest.TEST_STRING	),
		
		// Test number 1	
		(	StringToTest		:= 'Hello',
		  	WStringToTest 		:= "Hello",
			StringToContain 	:= 'h',
			WStringToContain	:= "h",
			IgnoreCases			:= TRUE,
			Trim 				:= FALSE,
			ExpectedResult  	:= FALSE,
			typeToTest      	:= TypeToTest.TEST_WSTRING	),
		
		// Test number 2	
		(	StringToTest		:= 'Hello',
		  	WStringToTest 		:= "Hello",
			StringToContain 	:= 'h',
			WStringToContain	:= "h",
			IgnoreCases			:= FALSE,
			Trim 				:= FALSE,
			ExpectedResult  	:= TRUE,
			typeToTest      	:= TypeToTest.TEST_STRING	),

		// Test number 3			
		(	StringToTest		:= 'Hello',
		  	WStringToTest 		:= "Hello",
			StringToContain 	:= 'h',
			WStringToContain	:= "h",
			IgnoreCases			:= FALSE,
			Trim 				:= FALSE,
			ExpectedResult  	:= TRUE,
			typeToTest      	:= TypeToTest.TEST_WSTRING	),
			
		// Test number 4	
		(	StringToTest		:= ' Hello',
		  	WStringToTest 		:= " Hello",
			StringToContain 	:= 'H',
			WStringToContain	:= "H",
			IgnoreCases			:= FALSE,
			Trim 				:= TRUE,
			ExpectedResult  	:= FALSE,
			typeToTest      	:= TypeToTest.TEST_STRING	),

		// Test number 5			
		(	StringToTest		:= ' Hello',
		  	WStringToTest 		:= " Hello",
			StringToContain 	:= 'H',
			WStringToContain	:= "H",
			IgnoreCases			:= FALSE,
			Trim 				:= TRUE,
			ExpectedResult  	:= FALSE,
			typeToTest      	:= TypeToTest.TEST_WSTRING	),
			
		// Test number 6	
		(	StringToTest		:= 'Kind and evil',
		  	WStringToTest 		:= "Добро и зло",
			StringToContain 	:= 'Kind',
			WStringToContain	:= "Добро",
			IgnoreCases			:= FALSE,
			Trim 				:= FALSE,
			ExpectedResult  	:= FALSE,
			typeToTest      	:= TypeToTest.TEST_STRING	),

		// Test number 7			
		(	StringToTest		:= 'Kind and evil',
		  	WStringToTest 		:= "Добро и зло",
			StringToContain 	:= 'Kind',
			WStringToContain	:= "Добро",
			IgnoreCases			:= FALSE,
			Trim 				:= FALSE,
			ExpectedResult  	:= FALSE,
			typeToTest      	:= TypeToTest.TEST_WSTRING	),
			
		// Test number 8	
		(	StringToTest		:= 'Kind and evil',
		  	WStringToTest 		:= "Добро и зло",
			StringToContain 	:= 'ind',
			WStringToContain	:= "обро",
			IgnoreCases			:= FALSE,
			Trim 				:= FALSE,
			ExpectedResult  	:= TRUE,
			typeToTest      	:= TypeToTest.TEST_STRING	),

		// Test number 9			
		(	StringToTest		:= 'Kind and evil',
		  	WStringToTest 		:= "Добро и зло",
			StringToContain 	:= 'ind',
			WStringToContain	:= "обро",
			IgnoreCases			:= FALSE,
			Trim 				:= FALSE,
			ExpectedResult  	:= TRUE,
			typeToTest      	:= TypeToTest.TEST_WSTRING	),
			
		// Test number 10	
		(	StringToTest		:= 'Kind and evil',
		  	WStringToTest 		:= "Добро и зло",
			StringToContain 	:= 'Kind',
			WStringToContain	:= "добро",
			IgnoreCases			:= TRUE,
			Trim 				:= FALSE,
			ExpectedResult  	:= FALSE,
			typeToTest      	:= TypeToTest.TEST_STRING	),

		// Test number 11			
		(	StringToTest		:= 'Kind and evil',
		  	WStringToTest 		:= "Добро и зло",
			StringToContain 	:= 'Kind',
			WStringToContain	:= "добро",
			IgnoreCases			:= TRUE,
			Trim 				:= FALSE,
			ExpectedResult  	:= FALSE,
			typeToTest      	:= TypeToTest.TEST_WSTRING	),
			
		// Test number 12	
		(	StringToTest		:= ' Kind and evil',
		  	WStringToTest 		:= " Добро и зло",
			StringToContain 	:= 'Kind',
			WStringToContain	:= "добро",
			IgnoreCases			:= TRUE,
			Trim 				:= TRUE,
			ExpectedResult  	:= FALSE,
			typeToTest      	:= TypeToTest.TEST_STRING	),

		// Test number 13			
		(	StringToTest		:= ' Kind and evil',
		  	WStringToTest 		:= " Добро и зло",
			StringToContain 	:= 'Kind',
			WStringToContain	:= "добро",
			IgnoreCases			:= TRUE,
			Trim 				:= TRUE,
			ExpectedResult  	:= FALSE,
			typeToTest      	:= TypeToTest.TEST_WSTRING	),
			
		// Test number 14			
		(	StringToTest		:= '',
		  	WStringToTest 		:= " 🧛",
			StringToContain 	:= '',
			WStringToContain	:= "🧛",
			IgnoreCases			:= TRUE,
			Trim 				:= TRUE,
			ExpectedResult  	:= FALSE,
			typeToTest      	:= TypeToTest.TEST_WSTRING	),
			
		// Test number 15			
		(	StringToTest		:= '',
		  	WStringToTest 		:= " 🧛",
			StringToContain 	:= '',
			WStringToContain	:= "🧛",
			IgnoreCases			:= TRUE,
			Trim 				:= FALSE,
			ExpectedResult  	:= TRUE,
			typeToTest      	:= TypeToTest.TEST_WSTRING	),

		// Test number 16			
		(	StringToTest		:= '',
		  	WStringToTest 		:= "🧛",
			StringToContain 	:= '',
			WStringToContain	:= "🧛",
			IgnoreCases			:= FALSE,
			Trim 				:= FALSE,
			ExpectedResult  	:= FALSE,
			typeToTest      	:= TypeToTest.TEST_WSTRING	),
			
		// Test number 17			
		(	StringToTest		:= ' hello world ',
		  	WStringToTest 		:= " hello world ",
			StringToContain 	:= '  ',
			WStringToContain	:= "  ",
			IgnoreCases			:= TRUE,
			Trim 				:= FALSE,
			ExpectedResult  	:= TRUE,
			typeToTest      	:= TypeToTest.TEST_WSTRING	),

		// Test number 18			
		(	StringToTest		:= ' hello world ',
		  	WStringToTest 		:= " hello world ",
			StringToContain 	:= '  ',
			WStringToContain	:= "  ",
			IgnoreCases			:= TRUE,
			Trim 				:= FALSE,
			ExpectedResult  	:= TRUE,
			typeToTest      	:= TypeToTest.TEST_STRING	)
					

	];
END_VAR

// ---- Version/Global_Version.TcGVL
{attribute 'TcGenerated'}
{attribute 'no-analysis'}
{attribute 'linkalways'}
// This function has been automatically generated from the project information.
VAR_GLOBAL CONSTANT
	{attribute 'const_non_replaced'}
	stLibVersion_CNM_AssertionInterfaceTests : ST_LibVersion := (iMajor := 1, iMinor := 0, iBuild := 0, iRevision := 47, nFlags := 0, sVersion := '1.0.0.47');
END_VAR

// ---- AssertionTester/AssertionResult/interfaces/IAssertorContainer.TcIO
(*

short summary
=============
An assertion is handled internally, and there is no common way to determine if an assertion was wrong.
This interface is just a helper to build containers to test assertions in a unified way.

.. <legal notes>

legal notes
=================
| SPDX-FileCopyrightText: © 2023 ekvip automation GmbH <info@ekvip.de>
| SPDX-License-Identifier: Apache-2.0
| For details check: Apache-2.0_

.. _Apache-2.0: https://www.apache.org/licenses/LICENSE-2.0

.. </legal notes>

properties
==========

*)

INTERFACE IAssertorContainer //EXTENDS CNM_AbstractObject.IObject

PROPERTY assertor :CNM_AssertionInterfaceLib.IAssertor
GET
END_GET
END_PROPERTY

METHOD resetAssertor
VAR_INPUT
END_VAR
END_METHOD

(*

short summary
=============
This property is used by the tests to determine if the assertion was right or wrong (getter)

.. <legal notes>

legal notes
=================
| SPDX-FileCopyrightText: © 2022 ekvip automation GmbH <info@ekvip.de>
| SPDX-License-Identifier: Apache-2.0
| For details check: Apache-2.0_

.. _Apache-2.0: https://www.apache.org/licenses/LICENSE-2.0

.. </legal notes>

*)

PROPERTY wasAssertionWrong :BOOL
GET
END_GET
END_PROPERTY

END_INTERFACE

// ---- AssertionTester/interfaces/IAttachAssertorContainer.TcIO
(*

short summary
=============

.. <legal notes>

legal notes
=================
| SPDX-FileCopyrightText: © 2023 ekvip automation GmbH <info@ekvip.de>
| SPDX-License-Identifier: Apache-2.0
| For details check: Apache-2.0_

.. _Apache-2.0: https://www.apache.org/licenses/LICENSE-2.0

.. </legal notes>

*)

{warning 'header is generated please add your documentation'}
INTERFACE IAttachAssertorContainer EXTENDS  __SYSTEM.IQueryInterface

(*

short summary
=============

.. <legal notes>

legal notes
=================
| SPDX-FileCopyrightText: © 2023 ekvip automation GmbH <info@ekvip.de>
| SPDX-License-Identifier: Apache-2.0
| For details check: Apache-2.0_

.. _Apache-2.0: https://www.apache.org/licenses/LICENSE-2.0

.. </legal notes>

*)

{warning 'header is generated please add your documentation'}
PROPERTY attachAssertorContainer : IAssertorContainer
SET
END_SET
END_PROPERTY

END_INTERFACE

// ---- AssertionTester/AssertionTests/BinaryAssertions/classes/BinaryAssertionsTests.TcPOU
(*

short summary
==================
This class tests all methods of binary assertions
with various combinations of inputs and checks expected 
outputs are satisfied or not

.. <legal notes>

legal notes
=================
| SPDX-FileCopyrightText: © 2022 ekvip automation GmbH <info@ekvip.de>
| SPDX-License-Identifier: Apache-2.0
| For details check: Apache-2.0_

.. _Apache-2.0: https://www.apache.org/licenses/LICENSE-2.0

.. </legal notes>

methods and properties
======================

*)

FUNCTION_BLOCK BinaryAssertionsTests EXTENDS AbstractAssertorTest
VAR_INPUT
	(* shall be not set, because this is for the null pointer edge case tests *)
	NULL :ANY;
END_VAR
VAR
	(* boolean value TRUE *)
	BOOLEAN_TRUE							:BOOL := TRUE;
	(* boolean value FALSE *)
	BOOLEAN_FALSE							:BOOL := FALSE;
	(* long word value one *)
	LWORD_WITH_VALUE_1						:LWORD := 16#0000_0000_0000_0000_0000_0000_0000_0001;
	(* word value 255 *)
	ALL_BITS_SET_AT_LOW_BYTE				:WORD := 16#00FF;
	(* double word vaule 255 *)
	ALL_BITS_SET_AT_LOW_BYTE_DWORD			:DWORD := 16#0000_00FF;
	(* double word value 16#FF00_FF00 *)
	NO_BITS_SET_AT_MID_BYTES				:DWORD := 16#FF00_00FF;
	(* byte array [0..299] all zero *)
	BYTE_ARRAY_ALL_BYTES_ZERO				:ARRAY[0..299] OF BYTE := [300(0)];
	(* byte array [0..299] 100 zero, 100 16#FF, 100 zero *)
	BYTE_ARRAY_MID_BYTES_FF_ONLY			:ARRAY[0..299] OF BYTE := [100(0),100(16#FF),100(0)];
	(* byte array with two dimensions [0..2][0..99] all zero *)
	ARRAY_OF_BYTE_ARRAY_ALL_BYTES_ZERO		:ARRAY[0..2] OF ARRAY[0..99] OF BYTE := [[100(0)],[100(0)],[100(0)]];	
END_VAR
VAR CONSTANT	
	(* prefix to unify the test names *)
	TEST_NAME_PREFIX						:STRING := 'assert.binary.';
END_VAR

THIS^.runIsEqualToTests();
THIS^.runIsNotEqualToTests();
THIS^.runIsGreaterThanTests();
THIS^.runIsLessThanTests();

(*

short summary
==================
This test method is a helper function to create a unified test name

.. <legal notes>

legal notes
=================
| SPDX-FileCopyrightText: © 2022 ekvip automation GmbH <info@ekvip.de>
| SPDX-License-Identifier: Apache-2.0
| For details check: Apache-2.0_

.. _Apache-2.0: https://www.apache.org/licenses/LICENSE-2.0

.. </legal notes>

parameters
==========

*)

METHOD PROTECTED getTestNameFor :Tc2_System.T_MaxString
VAR_INPUT
	(* name of the method to test, to create a unified test name *)
	nameOfMethodToTest	:Tc2_System.T_MaxString;
END_VAR
getTestNameFor := Tc2_Standard.CONCAT(THIS^.TEST_NAME_PREFIX, nameOfMethodToTest);
END_METHOD

(*

short summary
==================
This test method tests ``assert.binary.isEqualTo``
method of CNM_AssertionInterfaceLib library with various inputs

.. <legal notes>

legal notes
=================
| SPDX-FileCopyrightText: © 2022 ekvip automation GmbH <info@ekvip.de>
| SPDX-License-Identifier: Apache-2.0
| For details check: Apache-2.0_

.. _Apache-2.0: https://www.apache.org/licenses/LICENSE-2.0

.. </legal notes>

*)

METHOD runIsEqualToTests
RETURN (NOT TcUnit.TEST_ORDERED(THIS^.getTestNameFor('isEqualTo')));

THIS^.testIsEqualTo(
	data			:= THIS^.BOOLEAN_FALSE,
	dataToCompare	:= THIS^.BOOLEAN_FALSE,
	assertionIsWrong:= FALSE,
	testDataInfo	:= 'data is a boolean FALSE, dataToCompare is a aboolean FALSE'
);

THIS^.testIsEqualTo(
	data			:= THIS^.BOOLEAN_TRUE,
	dataToCompare	:= THIS^.BOOLEAN_FALSE,
	assertionIsWrong:= TRUE,
	testDataInfo	:= 'data is a boolean TRUE, dataToCompare is a boolean FALSE'
);

THIS^.testIsEqualTo(
	data			:= THIS^.BOOLEAN_TRUE,
	dataToCompare	:= NULL,
	assertionIsWrong:= TRUE,
	testDataInfo	:= 'data is a boolean TRUE, dataToCompare is null'
);

THIS^.testIsEqualTo(
	data			:= NULL,
	dataToCompare	:= NULL,
	assertionIsWrong:= FALSE,
	testDataInfo	:= 'data is null, dataToCompare is null'
);

THIS^.testIsEqualTo(
	data			:= THIS^.BYTE_ARRAY_ALL_BYTES_ZERO,
	dataToCompare	:= THIS^.BOOLEAN_FALSE,
	assertionIsWrong:= FALSE,
	testDataInfo	:= 'data is a byte array [300(0)], dataToCompare is a boolean FALSE'
);

THIS^.testIsEqualTo(
	data			:= THIS^.BYTE_ARRAY_ALL_BYTES_ZERO,
	dataToCompare	:= THIS^.ARRAY_OF_BYTE_ARRAY_ALL_BYTES_ZERO,
	assertionIsWrong:= FALSE,
	testDataInfo	:= 'data is a byte array [300(0)], dataToCompare is a byte array [[100(0)],[100(0)],[100(0)]]'
);

THIS^.testIsEqualTo(
	data			:= THIS^.BYTE_ARRAY_MID_BYTES_FF_ONLY,
	dataToCompare	:= THIS^.ARRAY_OF_BYTE_ARRAY_ALL_BYTES_ZERO,
	assertionIsWrong:= TRUE,
	testDataInfo	:= 'data is a byte array [100(0),100(16#FF),100(0)], dataToCompare is a byte array [[100(0)],[100(0)],[100(0)]]'
);

THIS^.testIsEqualTo(
	data			:= THIS^.ALL_BITS_SET_AT_LOW_BYTE,
	dataToCompare	:= THIS^.ALL_BITS_SET_AT_LOW_BYTE_DWORD,
	assertionIsWrong:= FALSE,
	testDataInfo	:= 'data is a word 16#00FF, dataToCompare is dword 16#0000_00FF'
);

THIS^.testIsEqualTo(
	data			:= THIS^.ALL_BITS_SET_AT_LOW_BYTE_DWORD,
	dataToCompare	:= THIS^.ALL_BITS_SET_AT_LOW_BYTE,
	assertionIsWrong:= FALSE,
	testDataInfo	:= 'data is a dword 16#0000_00FF, dataToCompare is word 16#00FF'
);

THIS^.testIsEqualTo(
	data			:= THIS^.ALL_BITS_SET_AT_LOW_BYTE,
	dataToCompare	:= THIS^.NO_BITS_SET_AT_MID_BYTES,
	assertionIsWrong:= TRUE,
	testDataInfo	:= 'data is a word 16#00FF, dataToCompare is dword 16#FF00_00FF'
);

THIS^.testIsEqualTo(
	data			:= THIS^.NO_BITS_SET_AT_MID_BYTES,
	dataToCompare	:= THIS^.ALL_BITS_SET_AT_LOW_BYTE,
	assertionIsWrong:= TRUE,
	testDataInfo	:= 'data is a dword 16#FF00_00FF, dataToCompare is word 16#00FF'
);

THIS^.testIsEqualTo(
	data			:= THIS^.LWORD_WITH_VALUE_1,
	dataToCompare	:= THIS^.BOOLEAN_TRUE,
	assertionIsWrong:= FALSE,
	testDataInfo	:= 'data is a lword 16#0000_0000_0000_0000_0000_0000_0000_0001, dataToCompare is bool TRUE'
);

THIS^.testIsEqualTo(
	data			:= THIS^.LWORD_WITH_VALUE_1,
	dataToCompare	:= THIS^.BOOLEAN_FALSE,
	assertionIsWrong:= TRUE,
	testDataInfo	:= 'data is a lword 16#0000_0000_0000_0000_0000_0000_0000_0001, dataToCompare is bool FALSE'
);

TcUnit.TEST_FINISHED();
END_METHOD

(*

short summary
==================
This test method tests ``assert.binary.isGreaterThan``
method of CNM_AssertionInterfaceLib library with various inputs

.. <legal notes>

legal notes
=================
| SPDX-FileCopyrightText: © 2022 ekvip automation GmbH <info@ekvip.de>
| SPDX-License-Identifier: Apache-2.0
| For details check: Apache-2.0_

.. _Apache-2.0: https://www.apache.org/licenses/LICENSE-2.0

.. </legal notes>

*)

METHOD runIsGreaterThanTests
RETURN (NOT TcUnit.TEST_ORDERED(THIS^.getTestNameFor('isGreaterThan')));

THIS^.testIsGreaterThan(
	data			:= THIS^.BOOLEAN_FALSE,
	dataToCompare	:= THIS^.BOOLEAN_FALSE,
	assertionIsWrong:= TRUE,
	testDataInfo	:= 'data is a boolean FALSE, dataToCompare is a aboolean FALSE'
);

THIS^.testIsGreaterThan(
	data			:= THIS^.BOOLEAN_TRUE,
	dataToCompare	:= THIS^.BOOLEAN_FALSE,
	assertionIsWrong:= FALSE,
	testDataInfo	:= 'data is a boolean TRUE, dataToCompare is a boolean FALSE'
);

THIS^.testIsGreaterThan(
	data			:= THIS^.BOOLEAN_TRUE,
	dataToCompare	:= NULL,
	assertionIsWrong:= FALSE,
	testDataInfo	:= 'data is a boolean TRUE, dataToCompare is null'
);

THIS^.testIsGreaterThan(
	data			:= NULL,
	dataToCompare	:= NULL,
	assertionIsWrong:= TRUE,
	testDataInfo	:= 'data is null, dataToCompare is null'
);

THIS^.testIsGreaterThan(
	data			:= THIS^.BYTE_ARRAY_ALL_BYTES_ZERO,
	dataToCompare	:= THIS^.BOOLEAN_FALSE,
	assertionIsWrong:= TRUE,
	testDataInfo	:= 'data is a byte array [300(0)], dataToCompare is a boolean FALSE'
);

THIS^.testIsGreaterThan(
	data			:= THIS^.BYTE_ARRAY_ALL_BYTES_ZERO,
	dataToCompare	:= THIS^.ARRAY_OF_BYTE_ARRAY_ALL_BYTES_ZERO,
	assertionIsWrong:= TRUE,
	testDataInfo	:= 'data is a byte array [300(0)], dataToCompare is a byte array [[100(0)],[100(0)],[100(0)]]'
);

THIS^.testIsGreaterThan(
	data			:= THIS^.BYTE_ARRAY_MID_BYTES_FF_ONLY,
	dataToCompare	:= THIS^.ARRAY_OF_BYTE_ARRAY_ALL_BYTES_ZERO,
	assertionIsWrong:= FALSE,
	testDataInfo	:= 'data is a byte array [100(0),100(16#FF),100(0)], dataToCompare is a byte array [[100(0)],[100(0)],[100(0)]]'
);

THIS^.testIsGreaterThan(
	data			:= THIS^.ALL_BITS_SET_AT_LOW_BYTE,
	dataToCompare	:= THIS^.ALL_BITS_SET_AT_LOW_BYTE_DWORD,
	assertionIsWrong:= TRUE,
	testDataInfo	:= 'data is a word 16#00FF, dataToCompare is dword 16#0000_00FF'
);

THIS^.testIsGreaterThan(
	data			:= THIS^.ALL_BITS_SET_AT_LOW_BYTE_DWORD,
	dataToCompare	:= THIS^.ALL_BITS_SET_AT_LOW_BYTE,
	assertionIsWrong:= TRUE,
	testDataInfo	:= 'data is a dword 16#0000_00FF, dataToCompare is word 16#00FF'
);

THIS^.testIsGreaterThan(
	data			:= THIS^.ALL_BITS_SET_AT_LOW_BYTE,
	dataToCompare	:= THIS^.NO_BITS_SET_AT_MID_BYTES,
	assertionIsWrong:= TRUE,
	testDataInfo	:= 'data is a word 16#00FF, dataToCompare is dword 16#FF00_00FF'
);

THIS^.testIsGreaterThan(
	data			:= THIS^.NO_BITS_SET_AT_MID_BYTES,
	dataToCompare	:= THIS^.ALL_BITS_SET_AT_LOW_BYTE,
	assertionIsWrong:= FALSE,
	testDataInfo	:= 'data is a dword 16#FF00_00FF, dataToCompare is word 16#00FF'
);

THIS^.testIsGreaterThan(
	data			:= THIS^.LWORD_WITH_VALUE_1,
	dataToCompare	:= THIS^.BOOLEAN_TRUE,
	assertionIsWrong:= TRUE,
	testDataInfo	:= 'data is a lword 16#0000_0000_0000_0000_0000_0000_0000_0001, dataToCompare is bool TRUE'
);

THIS^.testIsGreaterThan(
	data			:= THIS^.LWORD_WITH_VALUE_1,
	dataToCompare	:= THIS^.BOOLEAN_FALSE,
	assertionIsWrong:= FALSE,
	testDataInfo	:= 'data is a lword 16#0000_0000_0000_0000_0000_0000_0000_0001, dataToCompare is bool FALSE'
);

THIS^.testIsGreaterThan(
	data			:= THIS^.BOOLEAN_TRUE,
	dataToCompare	:= THIS^.LWORD_WITH_VALUE_1,
	assertionIsWrong:= TRUE,
	testDataInfo	:= 'data is a bool TRUE, dataToCompare is bool 16#0000_0000_0000_0000_0000_0000_0000_0001'
);

THIS^.testIsGreaterThan(
	data			:= THIS^.BOOLEAN_FALSE,
	dataToCompare	:= THIS^.LWORD_WITH_VALUE_1,
	assertionIsWrong:= TRUE,
	testDataInfo	:= 'data is a bool FALSE, dataToCompare is bool 16#0000_0000_0000_0000_0000_0000_0000_0001'
);

TcUnit.TEST_FINISHED();
END_METHOD

(*

short summary
==================
This test method tests ``assert.binary.isLessThan``
method of CNM_AssertionInterfaceLib library with various inputs

.. <legal notes>

legal notes
=================
| SPDX-FileCopyrightText: © 2022 ekvip automation GmbH <info@ekvip.de>
| SPDX-License-Identifier: Apache-2.0
| For details check: Apache-2.0_

.. _Apache-2.0: https://www.apache.org/licenses/LICENSE-2.0

.. </legal notes>

*)

METHOD runIsLessThanTests
RETURN (NOT TcUnit.TEST_ORDERED(THIS^.getTestNameFor('isLessThan')));

THIS^.testIsLessThan(
	data			:= THIS^.BOOLEAN_FALSE,
	dataToCompare	:= THIS^.BOOLEAN_FALSE,
	assertionIsWrong:= TRUE,
	testDataInfo	:= 'data is a boolean FALSE, dataToCompare is a aboolean FALSE'
);

THIS^.testIsLessThan(
	data			:= THIS^.BOOLEAN_TRUE,
	dataToCompare	:= THIS^.BOOLEAN_FALSE,
	assertionIsWrong:= TRUE,
	testDataInfo	:= 'data is a boolean TRUE, dataToCompare is a boolean FALSE'
);

THIS^.testIsLessThan(
	data			:= THIS^.BOOLEAN_FALSE,
	dataToCompare	:= THIS^.BOOLEAN_TRUE,
	assertionIsWrong:= FALSE,
	testDataInfo	:= 'data is a boolean FALSE, dataToCompare is a boolean TRUE'
);

THIS^.testIsLessThan(
	data			:= THIS^.BOOLEAN_TRUE,
	dataToCompare	:= NULL,
	assertionIsWrong:= TRUE,
	testDataInfo	:= 'data is a boolean TRUE, dataToCompare is null'
);

THIS^.testIsLessThan(
	data			:= NULL,
	dataToCompare	:= THIS^.BOOLEAN_TRUE,
	assertionIsWrong:= FALSE,
	testDataInfo	:= 'data is null, dataToCompare is a boolean TRUE'
);

THIS^.testIsLessThan(
	data			:= NULL,
	dataToCompare	:= NULL,
	assertionIsWrong:= TRUE,
	testDataInfo	:= 'data is null, dataToCompare is null'
);

THIS^.testIsLessThan(
	data			:= THIS^.BYTE_ARRAY_ALL_BYTES_ZERO,
	dataToCompare	:= THIS^.BOOLEAN_FALSE,
	assertionIsWrong:= TRUE,
	testDataInfo	:= 'data is a byte array [300(0)], dataToCompare is a boolean FALSE'
);

THIS^.testIsLessThan(
	data			:= THIS^.BYTE_ARRAY_ALL_BYTES_ZERO,
	dataToCompare	:= THIS^.ARRAY_OF_BYTE_ARRAY_ALL_BYTES_ZERO,
	assertionIsWrong:= TRUE,
	testDataInfo	:= 'data is a byte array [300(0)], dataToCompare is a byte array [[100(0)],[100(0)],[100(0)]]'
);

THIS^.testIsLessThan(
	data			:= THIS^.ARRAY_OF_BYTE_ARRAY_ALL_BYTES_ZERO,
	dataToCompare	:= THIS^.BYTE_ARRAY_ALL_BYTES_ZERO,
	assertionIsWrong:= TRUE,
	testDataInfo	:= 'data is a byte array [100(0),100(0),100(0)], dataToCompare is a byte array [300(0)]'
);

THIS^.testIsLessThan(
	data			:= THIS^.BYTE_ARRAY_MID_BYTES_FF_ONLY,
	dataToCompare	:= THIS^.ARRAY_OF_BYTE_ARRAY_ALL_BYTES_ZERO,
	assertionIsWrong:= TRUE,
	testDataInfo	:= 'data is a byte array [100(0),100(16#FF),100(0)], dataToCompare is a byte array [[100(0)],[100(0)],[100(0)]]'
);

THIS^.testIsLessThan(
	data			:= THIS^.ARRAY_OF_BYTE_ARRAY_ALL_BYTES_ZERO,
	dataToCompare	:= THIS^.BYTE_ARRAY_MID_BYTES_FF_ONLY,
	assertionIsWrong:= FALSE,
	testDataInfo	:= 'data is a byte array [[100(0)],[100(0)],[100(0)]], dataToCompare is a byte array [100(0),100(16#FF),100(0)]'
);

THIS^.testIsLessThan(
	data			:= THIS^.ALL_BITS_SET_AT_LOW_BYTE_DWORD,
	dataToCompare	:= THIS^.ALL_BITS_SET_AT_LOW_BYTE,
	assertionIsWrong:= TRUE,
	testDataInfo	:= 'data is a dword 16#0000_00FF, dataToCompare is word 16#00FF'
);

THIS^.testIsLessThan(
	data			:= THIS^.ALL_BITS_SET_AT_LOW_BYTE,
	dataToCompare	:= THIS^.NO_BITS_SET_AT_MID_BYTES,
	assertionIsWrong:= FALSE,
	testDataInfo	:= 'data is a word 16#00FF, dataToCompare is dword 16#FF00_00FF'
);

THIS^.testIsLessThan(
	data			:= THIS^.NO_BITS_SET_AT_MID_BYTES,
	dataToCompare	:= THIS^.ALL_BITS_SET_AT_LOW_BYTE,
	assertionIsWrong:= TRUE,
	testDataInfo	:= 'data is a dword 16#FF00_00FF, dataToCompare is word 16#00FF'
);

THIS^.testIsLessThan(
	data			:= THIS^.LWORD_WITH_VALUE_1,
	dataToCompare	:= THIS^.BOOLEAN_TRUE,
	assertionIsWrong:= TRUE,
	testDataInfo	:= 'data is a lword 16#0000_0000_0000_0000_0000_0000_0000_0001, dataToCompare is bool TRUE'
);

THIS^.testIsLessThan(
	data			:= THIS^.LWORD_WITH_VALUE_1,
	dataToCompare	:= THIS^.BOOLEAN_FALSE,
	assertionIsWrong:= TRUE,
	testDataInfo	:= 'data is a lword 16#0000_0000_0000_0000_0000_0000_0000_0001, dataToCompare is bool FALSE'
);

THIS^.testIsLessThan(
	data			:= THIS^.BOOLEAN_TRUE,
	dataToCompare	:= THIS^.LWORD_WITH_VALUE_1,
	assertionIsWrong:= TRUE,
	testDataInfo	:= 'data is a bool TRUE, dataToCompare is bool 16#0000_0000_0000_0000_0000_0000_0000_0001'
);

THIS^.testIsLessThan(
	data			:= THIS^.BOOLEAN_FALSE,
	dataToCompare	:= THIS^.LWORD_WITH_VALUE_1,
	assertionIsWrong:= FALSE,
	testDataInfo	:= 'data is a bool FALSE, dataToCompare is bool 16#0000_0000_0000_0000_0000_0000_0000_0001'
);

TcUnit.TEST_FINISHED();
END_METHOD

(*

short summary
==================
This test method tests ``assert.binary.isNotEqualTo``
method of CNM_AssertionInterfaceLib library with various inputs

.. <legal notes>

legal notes
=================
| SPDX-FileCopyrightText: © 2022 ekvip automation GmbH <info@ekvip.de>
| SPDX-License-Identifier: Apache-2.0
| For details check: Apache-2.0_

.. _Apache-2.0: https://www.apache.org/licenses/LICENSE-2.0

.. </legal notes>

*)

METHOD runIsNotEqualToTests
RETURN (NOT TcUnit.TEST_ORDERED(THIS^.getTestNameFor('isNotEqualTo')));

THIS^.testIsNotEqualTo(
	data			:= THIS^.BOOLEAN_FALSE,
	dataToCompare	:= THIS^.BOOLEAN_FALSE,
	assertionIsWrong:= TRUE,
	testDataInfo	:= 'data is a boolean FALSE, dataToCompare is a aboolean FALSE'
);

THIS^.testIsNotEqualTo(
	data			:= THIS^.BOOLEAN_TRUE,
	dataToCompare	:= THIS^.BOOLEAN_FALSE,
	assertionIsWrong:= FALSE,
	testDataInfo	:= 'data is a boolean TRUE, dataToCompare is a boolean FALSE'
);

THIS^.testIsNotEqualTo(
	data			:= THIS^.BOOLEAN_TRUE,
	dataToCompare	:= NULL,
	assertionIsWrong:= FALSE,
	testDataInfo	:= 'data is a boolean TRUE, dataToCompare is null'
);

THIS^.testIsNotEqualTo(
	data			:= NULL,
	dataToCompare	:= NULL,
	assertionIsWrong:= TRUE,
	testDataInfo	:= 'data is null, dataToCompare is null'
);

THIS^.testIsNotEqualTo(
	data			:= THIS^.BYTE_ARRAY_ALL_BYTES_ZERO,
	dataToCompare	:= THIS^.BOOLEAN_FALSE,
	assertionIsWrong:= TRUE,
	testDataInfo	:= 'data is a byte array [300(0)], dataToCompare is a boolean FALSE'
);

THIS^.testIsNotEqualTo(
	data			:= THIS^.BYTE_ARRAY_ALL_BYTES_ZERO,
	dataToCompare	:= THIS^.ARRAY_OF_BYTE_ARRAY_ALL_BYTES_ZERO,
	assertionIsWrong:= TRUE,
	testDataInfo	:= 'data is a byte array [300(0)], dataToCompare is a byte array [[100(0)],[100(0)],[100(0)]]'
);

THIS^.testIsNotEqualTo(
	data			:= THIS^.BYTE_ARRAY_MID_BYTES_FF_ONLY,
	dataToCompare	:= THIS^.ARRAY_OF_BYTE_ARRAY_ALL_BYTES_ZERO,
	assertionIsWrong:= FALSE,
	testDataInfo	:= 'data is a byte array [100(0),100(16#FF),100(0)], dataToCompare is a byte array [[100(0)],[100(0)],[100(0)]]'
);

THIS^.testIsNotEqualTo(
	data			:= THIS^.ALL_BITS_SET_AT_LOW_BYTE,
	dataToCompare	:= THIS^.ALL_BITS_SET_AT_LOW_BYTE_DWORD,
	assertionIsWrong:= TRUE,
	testDataInfo	:= 'data is a word 16#00FF, dataToCompare is dword 16#0000_00FF'
);

THIS^.testIsNotEqualTo(
	data			:= THIS^.ALL_BITS_SET_AT_LOW_BYTE_DWORD,
	dataToCompare	:= THIS^.ALL_BITS_SET_AT_LOW_BYTE,
	assertionIsWrong:= TRUE,
	testDataInfo	:= 'data is a dword 16#0000_00FF, dataToCompare is word 16#00FF'
);

THIS^.testIsNotEqualTo(
	data			:= THIS^.ALL_BITS_SET_AT_LOW_BYTE,
	dataToCompare	:= THIS^.NO_BITS_SET_AT_MID_BYTES,
	assertionIsWrong:= FALSE,
	testDataInfo	:= 'data is a word 16#00FF, dataToCompare is dword 16#FF00_00FF'
);

THIS^.testIsNotEqualTo(
	data			:= THIS^.NO_BITS_SET_AT_MID_BYTES,
	dataToCompare	:= THIS^.ALL_BITS_SET_AT_LOW_BYTE,
	assertionIsWrong:= FALSE,
	testDataInfo	:= 'data is a dword 16#FF00_00FF, dataToCompare is word 16#00FF'
);

THIS^.testIsNotEqualTo(
	data			:= THIS^.LWORD_WITH_VALUE_1,
	dataToCompare	:= THIS^.BOOLEAN_TRUE,
	assertionIsWrong:= TRUE,
	testDataInfo	:= 'data is a lword 16#0000_0000_0000_0000_0000_0000_0000_0001, dataToCompare is bool TRUE'
);

THIS^.testIsNotEqualTo(
	data			:= THIS^.LWORD_WITH_VALUE_1,
	dataToCompare	:= THIS^.BOOLEAN_FALSE,
	assertionIsWrong:= FALSE,
	testDataInfo	:= 'data is a lword 16#0000_0000_0000_0000_0000_0000_0000_0001, dataToCompare is bool FALSE'
);

TcUnit.TEST_FINISHED();
END_METHOD

(*

short summary
==================
This test method tests ``assert.binary.isEqualTo``
method of CNM_AssertionInterfaceLib library, 
it provides the possibility to handover test data via parameter 


.. <legal notes>

legal notes
=================
| SPDX-FileCopyrightText: © 2022 ekvip automation GmbH <info@ekvip.de>
| SPDX-License-Identifier: Apache-2.0
| For details check: Apache-2.0_

.. _Apache-2.0: https://www.apache.org/licenses/LICENSE-2.0

.. </legal notes>

parameters
==========

*)

METHOD testIsEqualTo 
VAR_INPUT
	(* for the test it's the parameter ``data`` *)
	data				:ANY;
	(* for the test it's the parameter ``dataToCompare`` *)
	dataToCompare		:ANY;
	(* just the expectation if the assertion to test must be worng or true *)
	assertionIsWrong	:BOOL;
	(* info string what the test does *)
	testDataInfo		:Tc2_System.T_MaxString;
END_VAR
VAR
	(* contains the format string for the test message *)
	message	:Tc2_System.T_MaxString;
END_VAR
THIS^.assertorContainer.resetAssertor();

message := SEL(
	assertionIsWrong,
	Tc2_Standard.CONCAT(testDataInfo, ' assertion must be TRUE'),
	Tc2_Standard.CONCAT(testDataInfo, ' assertion must be FALSE')
);

THIS^.assertorContainer.assertor.assert.binary.isEqualTo(
	data := data,
	dataToCompare := dataToCompare,
	message := ''
);

THIS^.AssertEquals_BOOL(
	Expected 	:= assertionIsWrong,
	Actual 		:= THIS^.assertorContainer.wasAssertionWrong,
	Message 	:= message
);
END_METHOD

(*

short summary
==================
This test method tests ``assert.binary.isGreaterThan``
method of CNM_AssertionInterfaceLib library, 
it provides the possibility to handover test data via parameter 


.. <legal notes>

legal notes
=================
| SPDX-FileCopyrightText: © 2022 ekvip automation GmbH <info@ekvip.de>
| SPDX-License-Identifier: Apache-2.0
| For details check: Apache-2.0_

.. _Apache-2.0: https://www.apache.org/licenses/LICENSE-2.0

.. </legal notes>

parameters
==========

*)

METHOD testIsGreaterThan 
VAR_INPUT
	(* for the test it's the parameter ``data`` *)
	data				:ANY;
	(* for the test it's the parameter ``dataToCompare`` *)
	dataToCompare		:ANY;
	(* just the expectation if the assertion to test must be worng or true *)
	assertionIsWrong	:BOOL;
	(* info string what the test does *)
	testDataInfo		:Tc2_System.T_MaxString;
END_VAR
VAR
	(* contains the format string for the test message *)
	message	:Tc2_System.T_MaxString;
END_VAR
THIS^.assertorContainer.resetAssertor();

message := SEL(
	assertionIsWrong,
	Tc2_Standard.CONCAT(testDataInfo, ' assertion must be TRUE'),
	Tc2_Standard.CONCAT(testDataInfo, ' assertion must be FALSE')
);

